// TwinCAT 3 PLC project PLC1
// ProgramVersion: 3.1.4026.24
// CompilerDefines: VISU_USEPROPERTYINFO
// libraries:
//   Tc2_Standard, * (Beckhoff Automation GmbH)
//   Tc2_System, * (Beckhoff Automation GmbH)
//   Tc2_TcpIp, * (Beckhoff Automation GmbH)
//   Tc2_Utilities, * (Beckhoff Automation GmbH)
//   VisuDialogs, * (System)
//   VisuSymbols,3.5.10.0,System
// project tree:
//   DUTs/ E_AutoStep.TcDUT (not stored), E_ControlMode.TcDUT, E_LogSev.TcDUT, E_MasterAutoStep.TcDUT, E_RobotConnState.TcDUT, ST_HmiMasterAuto.TcDUT, ST_HmiMasterAutoCfg.TcDUT, ST_HmiPiston.TcDUT (not stored), ST_HmiPistonAuto.TcDUT, ST_HmiPistonAutoCfg.TcDUT, ST_HmiRobot.TcDUT, ST_RobotParams.TcDUT, ST_LogEntry.TcDUT, E_LogFileState.TcDUT, ST_HmiLogFile.TcDUT, ST_HmiLogFileCfg.TcDUT
//   / GlobalTextList.TcGTLO, IOmapTask.TcTTO, PlcTask.TcTTO (not stored), VISU_TASK.TcTTO
//   GVLs/ GVL_App.TcGVL, GVL_HMI.TcGVL, GVL_HmiPersistent.TcGVL, GVL_IO.TcGVL (not stored), GVL_Log.TcGVL, GVL_Robot.TcGVL
//   POUs/ F_LogEvent.TcPOU, FB_PersistentAutoSave.TcPOU, FB_LogCsvWriter.TcPOU, FB_MasterAutoCycle.TcPOU, FB_PistonAutoCycle.TcPOU (not stored), FB_RobotTcpClient.TcPOU, FB_SolSolPiston_2Pos.TcPOU, FB_SolSpringPiston_2Pos.TcPOU, MAIN.TcPOU, PRG_IoMap.TcPOU
//   VISU/ Main.TcVIS, PistonsManual.TcVIS, Logs.TcVIS, Robot.TcVIS, GripperManual.TcVIS, Piston.TcVIS, AutoMain.TcVIS, AutoConfig.TcVIS, VisualizationManager.TcVMO (not stored)
// real-time tasks:
//   TASK IOmapTask: cycle T#5ms, priority 15, ADS port 350
//   TASK PlcTask: cycle T#10ms, priority 20, ADS port 351
//   TASK VISU_TASK: cycle T#200000us, priority 30, ADS port 352
// I/O:
//   DEVICE Device 1 (EtherCAT), AmsNetId 5.79.93.36.2.1
//     Term 1 (EK1100) [EK1100 EtherCAT Coupler (2A E-Bus)]
//       Term 2 (EL1809) [EL1809 16Ch. Dig. Input 24V, 3ms]
//       Term 3 (EL1008) [EL1008 8Ch. Dig. Input 24V, 3ms]
//       Term 4 (EL2809) [EL2809 16Ch. Dig. Output 24V, 0.5A]
//       Term 5 (EL9011) [EL9011 End Terminal]
// variable links:
//   PLC1/PLC1 Instance <-> Device 1 (EtherCAT)/Term 1 (EK1100)/Term 2 (EL1809)
//     IOmapTask Inputs/GVL_IO.dIn[{1..16}] <-> Channel {1..16}/Input  (16 links)
//   PLC1/PLC1 Instance <-> Device 1 (EtherCAT)/Term 1 (EK1100)/Term 3 (EL1008)
//     IOmapTask Inputs/GVL_IO.dIn[{17..24}] <-> Channel {1..8}/Input  (8 links)
//   PLC1/PLC1 Instance <-> Device 1 (EtherCAT)/Term 1 (EK1100)/Term 4 (EL2809)
//     IOmapTask Outputs/GVL_IO.dOut[{1..16}] <-> Channel {1..16}/Output  (16 links)

CONFIGURATION PLC1
    RESOURCE PLC ON TwinCAT3
        TASK IOmapTask(INTERVAL := T#5ms, PRIORITY := 15);
        TASK VISU_TASK(INTERVAL := T#200000us, PRIORITY := 30);
        PROGRAM PRG_IoMap WITH IOmapTask : PRG_IoMap;
        PROGRAM VisuElems_Visu_Prg WITH VISU_TASK : VisuElems.Visu_Prg;
    END_RESOURCE
END_CONFIGURATION

// ---- DUTs/E_ControlMode.TcDUT
{attribute 'qualified_only'}
{attribute 'strict'}
{attribute 'to_string'}
TYPE E_ControlMode :
(
    Manual    := 0,
    Automatic := 1
) ;
END_TYPE

// ---- DUTs/E_LogSev.TcDUT
{attribute 'qualified_only'}
{attribute 'strict'}
{attribute 'to_string'}
TYPE E_LogSev :
(
    DBG   := 0,   // dropped by F_LogEvent when GVL_Log.bDebugMode = FALSE
    INFO  := 1,
    WARN  := 2,
    ERR   := 3
) ;
END_TYPE

// ---- DUTs/E_MasterAutoStep.TcDUT
{attribute 'qualified_only'}
{attribute 'strict'}
{attribute 'to_string'}
TYPE E_MasterAutoStep :
(
    IDLE                 := 0,
    SEP_EXTENDING        := 1,
    WAIT_POS2            := 2,
    PUSH_EXTENDING       := 3,
    DWELL_PUSH           := 4,
    PUSH_RETRACTING      := 5,
    PUSH_RETRACTED_DWELL := 6,
    SEP_RETRACTING       := 7,
    SEP_RETRACTED_DWELL  := 8,
    INIT_PUSH_RETRACTING := 10,
    INIT_SEP_RETRACTING  := 11,
    INIT_GRIP_RETRACTING := 12,
    // Renamed from WAIT_PLATE 2026-08-05. Wire value 20 is UNCHANGED, so the
    // robot cannot tell the difference; only the panel text and the source read
    // differently. It does more than wait -- it is the plate-presence gate.
    CHECK_PLATE          := 20,
    GRIP_EXTENDING       := 21,
    GRIP_RETRACTING      := 22,
    MANUAL               := 30,
    // In Automatic but NOT armed: the pistons have not been homed under
    // operator control since power-up / Manual / a STOP, so the robot must not
    // command a cycle. Exited only by an operator START (HMI button or PB3),
    // which runs the INIT retract chain and lands in IDLE.
    //
    // 40 sits in the same "not a sequence step" class as MANUAL(30) and
    // ERR(99). Values are WIRE values -- nStateOut is read by the robot -- so
    // nothing here may ever be renumbered.
    //
    // Keep the name short: sStepText is STRING(20) and INIT_PUSH_RETRACTING
    // already fills it exactly, so a longer enumerator would truncate.
    NOT_HOMED            := 40,

    // Fault-recovery retract chain, added 2026-08-05. Same MOTION as the
    // RETRACT/INIT chain (push, then sep, then grip -- the collision ordering)
    // but its own identity, so a failed recovery is distinguishable from a
    // failed arming: distinct sStepText, distinct error codes 12/13/14, and a
    // distinct value on the wire.
    //
    // Entered only from ERR on RESET; exits to IDLE (armed). 50/51/52 rather
    // than 13/14/15 because a fresh decade matches the convention that
    // non-bulb-cycle states own decades (30 Manual, 40 Not-homed, 99 Err), and
    // STATE:5x is instantly greppable in a robot log. Adjacency to 10/11/12
    // would invite exactly the confusion these states exist to remove.
    //
    // The robot needs NO new branch: it acts on 0 (armed), 99 (faulted) and
    // treats everything else as "wait", which is correct for all three.
    //
    // Names are <= 20 chars because sStepText is STRING(20).
    RECOVER_PUSH_RETR    := 50,
    RECOVER_SEP_RETR     := 51,
    RECOVER_GRIP_RETR    := 52,

    ERR                  := 99
) ;
END_TYPE

// ---- DUTs/E_RobotConnState.TcDUT
{attribute 'qualified_only'}
{attribute 'strict'}
{attribute 'to_string'}
TYPE E_RobotConnState :
(
    Disconnected := 0,
    Connecting   := 1,
    Connected    := 2,
    Error        := 3
) ;
END_TYPE

// ---- DUTs/ST_HmiMasterAuto.TcDUT
TYPE ST_HmiMasterAuto :
STRUCT
    // Display label ('MasterAuto'). Set from GVL_HMI init, never written by FB.
    Name             : STRING(30);

    // HMI writes -- momentary command buttons (R_TRIG inside FB latches the
    // rising edge). NOTE bStart means "home the pistons and arm", NOT "run a
    // bulb cycle" -- only the robot's CMD:1 starts a cycle. Also driven by the
    // green PB3 in Automatic (see MAIN).
    bStart           : BOOL;
    (* Operator "run ONE bulb from IDLE" -- the HMI parallel to holding the
       orange PB2 + green PB3 combo, and to the robot's CMD:1. Momentary:
       FB_MasterAutoCycle detects the rising edge and clears it.

       Deliberately a SEPARATE field from bStart. bStart means "home and
       arm" and is accepted in NOT_HOMED only; making it also mean "run a
       bulb" in IDLE would give one symbol two meanings that differ by
       state, which is exactly the shape that let a green-before-orange
       combo press silently lose its bulb request (fixed 2026-08-05 by
       removing START from IDLE -- do not put it back).

       Also separate from bSimStartAssembly, which is the documented BENCH
       stand-in for the robot. Two fields keep "an operator started a bulb"
       and "someone simulated the robot" distinguishable in the log ring. *)
    bStartCycle      : BOOL;
    bStop            : BOOL;
    bReset           : BOOL;

    // FB writes -- status.
    //
    // Defaults to NOT_HOMED, and that default is what keeps the machine still
    // after a power cycle: GVL_HMI is plain VAR_GLOBAL, so this initialiser is
    // re-applied on every cold boot and every download. bAutoMode persists, so
    // without it the panel would come back in Automatic reporting IDLE(0) and a
    // running robot could command a cycle with the pistons anywhere.
    eStep            : E_MasterAutoStep := E_MasterAutoStep.NOT_HOMED;
    sStepText        : STRING(20);   // human-readable mirror of eStep
    tElapsedS        : LREAL;        // seconds spent in the current step (0.0 on transition)
    iErrorCode       : INT;          // 0 = OK; see FB_MasterAutoCycle header for the code table
    sErrorText       : STRING(80);
    nCyclesCompleted : UDINT;        // incremented at end of GRIP_RETRACTING

    // HMI writes -- bench sim of the robot's start command. Rising edge inside
    // the FB behaves the same as an incoming CMD:1 pulse (see bExtStartPulse).
    // FB auto-clears this flag after the rising edge is consumed.
    bSimStartAssembly      : BOOL;

    // HMI writes -- per-step Simulate flags. Rising edge shortcuts the current
    // step's wait condition (FB clears the flag on consumption via R_TRIG.Q).
    bSimStep_Idle          : BOOL;
    bSimStep_InitPushRet   : BOOL;
    bSimStep_InitSepRet    : BOOL;
    bSimStep_InitGripRet   : BOOL;
    bSimStep_WaitPlate     : BOOL;
    bSimStep_GripExt       : BOOL;
    bSimStep_SepExt        : BOOL;
    bSimStep_WaitPos2      : BOOL;
    bSimStep_PushExt       : BOOL;
    bSimStep_DwellPush     : BOOL;
    bSimStep_PushRet       : BOOL;
    bSimStep_PushRetDwell  : BOOL;
    bSimStep_SepRet        : BOOL;
    bSimStep_SepRetDwell   : BOOL;
    bSimStep_GripRet       : BOOL;
    (* The RECOVER chain wants sim flags for the same reason the INIT chain
       has them: all three are sensor-waiting states, so without these a
       recovery cannot be stepped on a bench whose sensors are not wired.
       Added 2026-08-05; the RECOVER states themselves shipped without them. *)
    bSimStep_RecoverPushRet : BOOL;
    bSimStep_RecoverSepRet  : BOOL;
    bSimStep_RecoverGripRet : BOOL;
END_STRUCT
END_TYPE

// ---- DUTs/ST_HmiMasterAutoCfg.TcDUT
TYPE ST_HmiMasterAutoCfg :
STRUCT
    // Timers, milliseconds. UDINT so HMI NumericInput binds directly.
    tDwellPushMs            : UDINT := 2000;   // DWELL_PUSH -- hold at push-extended
    tPushRetractedDwellMs   : UDINT := 500;    // PUSH_RETRACTED_DWELL -- hold after push retract
    tSepRetractedDwellMs    : UDINT := 500;    // SEP_RETRACTED_DWELL -- hold after sep retract before IDLE

    // Timeout guards every non-DWELL waiting state. On expiry, iErrorCode is
    // set to the step's numeric code and the cycle enters ERR.
    tStepTimeoutMs          : UDINT := 10000;

    // Dedicated timeout for CHECK_PLATE (bounded by robot placement time, not
    // by a motion budget). On expiry, iErrorCode := 9 and the cycle enters ERR
    // — unless bBypassPlateSensors is set, see below.
    tPlateWaitTimeoutMs     : UDINT := 10000;

    // Panel push-button HOLD durations, milliseconds. Both are deliberate
    // two-hand / sustained gestures rather than edges, so a knock or a brushed
    // sleeve cannot trigger them.
    //
    // tPbStopHoldMs  — how long the RED PB1 must be held in Automatic to STOP
    //                  the machine (disarm to NOT_HOMED).
    // tPbStartHoldMs — how long the GREEN PB3 and ORANGE PB2 must be held
    //                  TOGETHER to start one bulb cycle from IDLE, which is the
    //                  operator's parallel to the robot's CMD:1.
    //
    // Editable on AutoMain so the duration can be tuned to the operators
    // without a rebuild.
    tPbStopHoldMs           : UDINT := 1000;
    tPbStartHoldMs          : UDINT := 1000;

    // If TRUE, the 4 movement states ignore sensor feedback and advance when
    // tStepTimeoutMs expires — the timeout doubles as the fixed step duration.
    // No timeout-error path while sensorless. Mirrors ST_HmiPistonAutoCfg.bNoSensors.
    // Deliberately does NOT cover WAIT_PLATE — use bBypassPlateSensors for that.
    bNoSensors              : BOOL  := FALSE;

    // Plate-sensor bypass. Removes only the WAIT_PLATE timeout ERROR, not the
    // wait itself: the bPlateSenL AND bPlateSenR fast-path still advances the
    // cycle as normal, so with healthy sensors nothing changes. With unwired
    // or faulty ones, tPlateWaitTimeoutMs degrades into a fixed placement
    // dwell and the cycle continues instead of raising error 9.
    // Separate from bNoSensors on purpose: skipping the plate gate is a
    // safety-relevant decision and should be made explicitly, not inherited
    // from a bench-testing flag.
    bBypassPlateSensors     : BOOL  := FALSE;

    // NOTE bAutoMode used to live here and does NOT any more (2026-08-06).
    // It moved to GVL_HMI.bAutoMode -- plain VAR_GLOBAL, initialised TRUE -- so
    // that every power-up comes back in Automatic instead of restoring whatever
    // mode the operator happened to leave selected. Persisting it was the older
    // decision (2026-07-27) and it had the property that a technician who
    // switched to Manual to jog a piston found the machine still in Manual after
    // a reboot; the machine's normal condition is Automatic, so that is now the
    // condition it boots into. It is safe because arming is separate: eStep still
    // defaults to NOT_HOMED, so nothing moves until someone presses ENABLE AUTO.
    //
    // This struct is now purely operator-tunable CONFIG -- timers and the two
    // bench flags -- which is also what makes it a coherent unit to put on its
    // own AutoConfig page.
END_STRUCT
END_TYPE

// ---- DUTs/ST_HmiPistonAuto.TcDUT
TYPE ST_HmiPistonAuto :
STRUCT
    // HMI writes — momentary commands (R_TRIG inside FB latches the rising edge)
    bStart : BOOL;
    bStop  : BOOL;
    bReset : BOOL;
    bAck   : BOOL;

    // FB writes — status (never touched by HMI)
    eStep            : E_AutoStep;
    sStepText        : STRING(20);   // human-readable mirror of eStep
    tElapsedS        : LREAL;        // seconds spent in the current step (0.0 on transition)
    bError           : BOOL;
    sErrorText       : STRING(80);
    nCyclesCompleted : UDINT;        // incremented at end of each DWELL_RET
END_STRUCT
END_TYPE

// ---- DUTs/ST_HmiPistonAutoCfg.TcDUT
TYPE ST_HmiPistonAutoCfg :
STRUCT
    // All times in milliseconds. UDINT so HMI NumericInput binds directly (no TIME<->UDINT juggling).

    // Dwell = how long to sit at the sensor before starting the reverse move.
    tDwellExtendedMs   : UDINT := 500;
    tDwellRetractedMs  : UDINT := 500;

    // Timeout = if we do not see the target sensor within this window, raise an error.
    tTimeoutExtendMs   : UDINT := 3000;
    tTimeoutRetractMs  : UDINT := 3000;

    // If TRUE, DWELL_RET loops back to EXTENDING instead of returning to IDLE.
    bContinuous        : BOOL  := FALSE;

    // If TRUE, the state machine ignores sensor feedback and advances on
    // timers alone: EXTENDING lasts tTimeoutExtendMs, RETRACTING lasts
    // tTimeoutRetractMs, then dwells run as usual. Use for bench cycling
    // when proximity switches aren't wired (SepSol2/3, PushSol2/3 today).
    // No feedback-mismatch check and no "sensor never arrived" error path.
    bNoSensors         : BOOL  := FALSE;
END_STRUCT
END_TYPE

// ---- DUTs/ST_HmiRobot.TcDUT
TYPE ST_HmiRobot :
STRUCT
    // Display label ('Robot'). Set from GVL_Robot, never written by bridge.
    Name           : STRING(30);

    // ------------------------------------------------------------------
    // Robot comms are now TCP-only. Start/reset commands come from the
    // robot as CMD:n replies (see ST_RobotParams.nRobotCmd); PLC state is
    // pushed to the robot as STATE:n (see ST_RobotParams.nStateOut). The
    // former discrete-I/O handshake (bStartAssembly/bAssemblyRunning wired
    // to STAND_SEQ_DO/STAND_SEQ_DI) is retired -- DI[13] and DO[7] are now
    // free channels.
    //
    // Fields below are the TCP status mirror written by FB_RobotTcpClient
    // and read by the HMI.
    // ------------------------------------------------------------------
    eConnState     : E_RobotConnState;
    sConnStateText : STRING(20);
    nPacketsRx     : UDINT;
    nPacketsTx     : UDINT;
    sLastMessage   : STRING(80);
    sLastTxMessage : STRING(80);

    // Consecutive failed connect attempts in the CURRENT outage; reset to 0 the
    // moment a connect succeeds. Added 2026-08-10 together with the edge guard on
    // the connect-failure log.
    //
    // THIS FIELD IS WHY THE SUPPRESSION IS SAFE. FB_RobotTcpClient re-dials every
    // ~3 s while bTcpEnable is TRUE, and it used to log an ERR every single time:
    // measured on the panel, all 20 slots of GVL_Log.aRecent were the same
    // 'Connect failed' line, and the Phase 2 CSV came out 95% that one message at
    // ~1.2 MB/day. Now only the first failure of an outage is logged (plus any
    // change of error NUMBER), so the information is not lost -- it moves here,
    // where the Robot page can show "312 failed attempts" in one field instead of
    // 312 log lines.
    nConnectFails  : UDINT;

    // The deprecated POS/AUTO_STARTED fields (bAtPos1/2/3, bTxAutoStarted,
    // bTxPushDone, bTxPistonsError, bRxResetError) were deleted 2026-07-26.
    // They existed only for legacy Flower_HMI page bindings on the retired
    // TCP POS protocol; that project is gone, no PLC code touched them, and
    // FlowerPyHmi does not poll them (scripts/check_pyhmi_contract.py).
END_STRUCT
END_TYPE

// ---- DUTs/ST_RobotParams.TcDUT
TYPE ST_RobotParams :
STRUCT
    // ------------------------------------------------------------------
    // Dobot tuning parameters exchanged over TCP:6001. TCP is now the ONLY
    // robot channel -- start/stop moved from discrete I/O to STATE:n / CMD:n
    // frames (see nStateOut / nRobotCmd below). Field names and order match
    // the robot's SYNC string (global.lua / dummy_server.py). Defaults
    // mirror the dummy server.
    //
    // UNITS AND RANGES. The four speeds are PERCENTAGES, not absolute
    // velocities: global.lua Init() passes J_SPEED / L_SPEED to VelJ() /
    // VelL(), and WAX_SPEED / WATER_SPEED feed the v= velocity-ratio option
    // of MovL. A global SpeedFactor(80) scales everything on top. The waits
    // are milliseconds. INT is an encoding detail, not a statement of range.
    //
    // Ranges below are the vendor's own -- the Dobot tuning GUI
    // (Robot\167-01-Saad\tcp client.py) clamps to them, and readme.txt
    // mirrors the table. The robot's Lua does NOT validate (src2.lua assigns
    // tonumber() straight through), so FB_RobotTcpClient.ClampParam enforces
    // them for every writer. The panel's NumericInputs also carry matching
    // InputBoxMin/Max, but per-control limits only bound their own control.
    // ------------------------------------------------------------------
    J_SPEED            : INT := 10;     //    1..100  %
    L_SPEED            : INT := 10;     //    1..100  %
    REPEATS            : INT := 2;      //    1..10
    START_WAIT         : INT := 500;    //   10..10000 ms
    WATER_WAIT         : INT := 500;    //   10..10000 ms
    STAND_WAIT         : INT := 2000;   //   10..10000 ms
    END_WAIT           : INT := 500;    //   10..10000 ms
    WATER_SPEED        : INT := 10;     //    0..100  %
    WAX_WAIT_TIME_IN   : INT := 500;    //    0..10000 ms
    WAX_WAIT_TIME_OUT  : INT := 500;    //   10..10000 ms
    WAX_SPEED          : INT := 10;     //    0..100  %

    // ------------------------------------------------------------------
    // Request flags -- FB_RobotTcpClient consumes each on the next idle
    // scan while Connected, sends the matching message, then auto-clears
    // the flag once the reply is received. Rising-level, not edge: setting
    // TRUE from the HMI is enough.
    // ------------------------------------------------------------------

    // Send GET_SYNC; the SYNC reply is parsed back into the 11 fields above.
    // The FB also raises this itself once, right after each (re)connect.
    bGetSync           : BOOL;

    // Raw escape hatch: send "sSetName:nSetVal" (e.g. "J_SPEED:15"); robot
    // replies "OK: SET NAME". NOT needed for the 11 params above -- writing
    // one of those fields directly (from the HMI or ST) is detected by
    // FB_RobotTcpClient's shadow-copy comparison and pushed automatically.
    // Use this only for names that are not fields of this struct.
    bSetParam          : BOOL;
    sSetName           : STRING(30);
    nSetVal            : INT;

    // Send "New_Bulb:1"; robot replies "OK: SET New_Bulb" and starts a fresh bulb.
    bTriggerNewBulb    : BOOL;

    // ------------------------------------------------------------------
    // State + command channel (replaces the retired discrete-I/O handshake).
    //
    // nStateOut : INT -- MAIN writes each scan. Value is TO_INT(eStep) in
    //   Automatic mode, or E_MasterAutoStep.MANUAL (30) when bAutoMode=FALSE.
    //   FB_RobotTcpClient sends "STATE:n" on change and every STATE_IDLE_MS
    //   as keep-alive.
    //
    // nRobotCmd : INT -- FB_RobotTcpClient writes each time a "CMD:n" reply
    //   carries a command. MAIN consumes it as a LEVEL (1 = start cycle,
    //   2 = reset error) and CLEARS it to 0 in the same scan; that clear is
    //   the PLC's acknowledgement, so the field normally reads 0 and a robot
    //   start is traced on the Logs page instead. The robot re-asserting the
    //   same value is therefore always honoured -- see the MAIN comment for
    //   the deadlock this replaced.
    // ------------------------------------------------------------------
    nStateOut          : INT;
    nRobotCmd          : INT;
END_STRUCT
END_TYPE

// ---- DUTs/ST_LogEntry.TcDUT
TYPE ST_LogEntry :
STRUCT
    // Wall-clock HH:MM:SS, stamped by F_LogEvent from GVL_Log.sNow (which
    // MAIN refreshes once a second from FB_LocalSystemTime). Added 2026-07-27
    // for the panel's Logs page, which has no drainer to stamp entries for it.
    //
    // This struct used to carry no timestamp on the reasoning that "Python
    // assigns wall-clock time when it drains the ring" — true, but that only
    // ever covered FlowerPyHmi. FlowerPyHmi still stamps its own arrival time
    // and ignores this field; the two do not have to agree, and sTime is the
    // more accurate of the two since it is taken at the moment of the event
    // rather than up to plc_ring_poll_ms later.
    //
    // Second resolution only. If sub-second ordering ever matters, add
    // nTick : UDINT rather than widening this string.
    sTime   : STRING(8);


    eSev    : E_LogSev;

    // Display mirror of eSev, set by F_LogEvent. Exists because the classic
    // VISU text output cannot resolve an enum to its enumerator name --
    // {attribute 'to_string'} only enables TO_STRING() in ST, it does not
    // teach the visualization anything. Same reason ST_HmiMasterAuto carries
    // sStepText next to eStep. FlowerPyHmi ignores this field; it renders
    // from eSev via its own SEV_NAMES map.
    // STRING(8), not STRING(4): the four current names top out at 4 chars,
    // but an exactly-sized string would silently truncate a longer one.
    sSevText : STRING(8);

    sSource : STRING(20);    // short instance name, e.g. 'SepSol1Auto'
    sMsg    : STRING(80);    // human-readable message
END_STRUCT
END_TYPE

// ---- DUTs/E_LogFileState.TcDUT
(*
   State of FB_LogCsvWriter (Phase 2 of docs/plans/log-csv-file.md).

   Declared in Phase 1, ahead of the FB that uses it, for the same reason the
   RECOVER_* wire values were reserved in one commit: the enum is the shared
   vocabulary between the PLC, the VISU page and FlowerPyHmi, so pinning the
   values once means the contract changes once.

   'to_string' is here for ST only. It does NOT make the classic VISU resolve an
   enumerator to its name -- that is settled in this project and is why
   ST_HmiLogFile carries an sStateText mirror. Binding eState to a VISU text
   output renders 0/1/2/3/4, which shipped wrong twice on the Logs page before
   being fixed on 2026-07-27.
*)
{attribute 'qualified_only'}
{attribute 'strict'}
{attribute 'to_string'}
TYPE E_LogFileState :
(
    // Logging disabled, or nothing pending. The resting state.
    OFF      := 0,

    // Entries buffered, waiting for the flush interval or a full buffer.
    BUFFER   := 10,

    // A flush is in flight. These three mirror the async chain rather than
    // being collapsed into one BUSY: if a write wedges, which of the three
    // it wedged in is the whole diagnostic, and there is no other way to see
    // it on a panel with no file viewer.
    OPENING  := 20,
    WRITING  := 21,
    CLOSING  := 22,

    // Rotation or retention work in progress (new day, size cap, or the
    // oldest-first delete sweep).
    ROTATING := 30,

    // A file operation failed. iErrorCode / sErrorText hold the detail and the
    // FB backs off on a timer rather than retrying every scan.
    FAILED   := 99
) ;
END_TYPE

// ---- DUTs/ST_HmiLogFile.TcDUT
(*
   Runtime status of the durable CSV log. Phase 1 of
   docs/plans/log-csv-file.md.

   Instanced as GVL_Log.stLogFile, i.e. VOLATILE -- GVL_Log is plain VAR_GLOBAL.
   That split is the point: the CONFIG persists (stLogFileCfg) and the STATUS
   does not. A persisted byte count or error text would be restored on the next
   boot describing a file the runtime has not opened, and a stale FAILED with a
   plausible error string is worse than no status at all.

   WHY THERE IS A STATUS STRUCT AT ALL. The CP6606 has no file viewer and no
   supported CPython, so nobody can look at the directory to see whether logging
   is working. Every question you would answer by looking at the filesystem has
   to be answerable from these fields instead: is it writing, to what, how big,
   how many files, has it lost anything, and if it stopped, why.
*)
TYPE ST_HmiLogFile :
STRUCT
    // Filename only, no directory -- sDir is already visible in the config and
    // repeating it here would just risk the two disagreeing.
    sCurrentFile      : STRING(40);

    // Bytes written to the current file. Compared against
    // uiMaxFileKB * 1024 to decide an in-day roll.
    uiBytesInFile     : UDINT;

    // CSV files currently in sDir, refreshed by the retention sweep.
    uiFilesOnDisk     : UDINT;

    // Entries the writer never got to see, because nWriteIdx advanced more than
    // the 256-slot ring holds while a flush was stalled.
    //
    // THIS FIELD IS THE WHOLE REASON THE DRAIN LOGIC IS ALLOWED TO SKIP. Losing
    // entries under a stall is unavoidable -- the ring is finite. Losing them
    // SILENTLY is not acceptable, so the count is published here and Phase 2
    // also emits one synthetic CSV row recording the gap, so the loss is visible
    // in the file itself and not only in a symbol nobody thought to read.
    udiEntriesDropped : UDINT;

    // Last file error. 0 = none. Latched until the next successful flush, so a
    // failure that has since cleared is still visible afterwards.
    iErrorCode        : UDINT;
    sErrorText        : STRING(80);

    eState            : E_LogFileState;

    // STRING mirror of eState. Required, not convenience: the classic VISU
    // cannot stringify an enum, so a text output bound to eState renders the
    // raw number. Every enum in this project carries such a mirror for exactly
    // this reason -- sStepText, sErrorText, sConnStateText, sSevText.
    sStateText        : STRING(12);
END_STRUCT
END_TYPE

// ---- DUTs/ST_HmiLogFileCfg.TcDUT
(*
   Operator-tunable config for the durable CSV log. Phase 1 of
   docs/plans/log-csv-file.md.

   Instanced as GVL_HmiPersistent.stLogFileCfg, i.e. VAR_GLOBAL PERSISTENT.
   Read the PERSISTENT DATA section of CLAUDE.md before adding a field here:
   PERSISTENT declares a durable storage CLASS, not an automatic save, and it is
   FB_PersistentAutoSave that actually flushes it ~2 s after edits stop. A new
   field is invisible to that FB until it is added to the shadow compare.

   COLD-BOOT DECISION, which CLAUDE.md requires for every new persistent field:
   NOTHING HERE IS CLEARED in MAIN's cold-boot block. Every field is operator or
   commissioning config, so surviving a power cycle is the entire point. Contrast
   the machine-state fields, where a persisted value can move pistons on power-up
   and which is why that block exists at all. Nothing here can start a motion.

   PER-FIELD COMMENTS IN THIS STRUCT MUST STAY SHORT -- put the prose in
   docs/plans/log-csv-file.md instead. This block, being the TYPE's comment, is
   free; a MEMBER's comment is not. TwinCAT ships a symbol's declaration comment
   inside its ADS symbol-info reply, and pyads' receive buffer is 798 bytes.
   sDir's original ~2.8 kB comment produced a 2967-byte reply, which fails
   symbol-info resolution -- and because read_list_by_name resolves every name
   in a sum-up up front, that took the field out of FlowerPyHmi's batched poll
   and onto an individual round trip: +88 ms on a 100 ms cycle, /events 3.3 Hz
   -> 2.62 Hz, measured against this panel 2026-08-12. FlowerPyHmi caps how many
   such symbols it will carry (5), and three others in this project are already
   spending that budget: GVL_HMI.bAutoMode (1400 B),
   GVL_Robot.stParams.nStateOut (991 B) and GVL_Robot.stRobot.nConnectFails
   (817 B).

   So the rule is not "write less"; it is "write it where an ADS client will not
   have to download it 10 times a second."
*)
TYPE ST_HmiLogFileCfg :
STRUCT
    // DEFAULT OFF, deliberately. The panel boots from Compact Flash and CF has
    // a finite erase budget -- the reason FB_PersistentAutoSave debounces its
    // own writes rather than saving on every keystroke. A machine that never
    // needs the file log should never spend flash on it, so writing to the card
    // is an explicit opt-in rather than something inherited from a download.
    bEnabled      : BOOL := FALSE;

    // Directory, WITH a trailing backslash; the writer appends the filename.
    // MUST stay under '\Hard Disk\': '\Temp\' and the device root are the WinCE
    // RAM object store and do not survive a restart. Never fall back to them.
    // Reasoning, measurements and the two rules: docs/plans/log-csv-file.md.
    // KEEP SHORT -- this comment ships in the ADS symbol-info reply (798 B cap);
    // oversized, it drops sDir out of FlowerPyHmi's batched poll. See below.
    sDir          : STRING(80) := '\Hard Disk\Logs\';

    // Roll to a new file part within the day if one file passes this. A guard
    // against a fault storm producing a single unwieldy file, not the primary
    // rotation trigger -- that is the date.
    uiMaxFileKB   : UDINT := 512;

    // Total ceiling for the directory. Phase 3 deletes oldest-first until the
    // sum is under this. 16 MB of INFO-level CSV is months of normal running.
    uiMaxTotalMB  : UDINT := 16;

    // Buffer flush interval. THE FLASH-WEAR CONTROL: entries accumulate in RAM
    // and reach the card once per interval, so a busy second costs one write
    // rather than dozens. Do not "improve" this into a write-per-entry -- that
    // is the change this comment exists to prevent.
    uiFlushSec    : UDINT := 10;
END_STRUCT
END_TYPE

// ---- GVLs/GVL_App.TcGVL
{attribute 'qualified_only'}
// Cooked IO aliases. Bound to the raw GVL_IO.dIn[i]/dOut[i] hardware arrays
// in MAIN's read-inputs / write-outputs bookends. No AT %*: these are plain
// BOOLs the FBs consume — the actual hardware wiring lives in GVL_IO.
//
// Tag convention: <Device>Sol<N>  = single EXTEND coil (SOL-Spring).
// The mechanical spring returns the actuator when the coil is de-energised,
// so no per-actuator Retract alias exists. DI still has a Retracted sensor.
//
//   SepSolN : Pin separator N   (DI 1..6, DO 1..3)
//   PushSolN: Pin push N        (DI 7..12, DO 4..6)
//   PbN / LedPbN: panel push buttons + status LEDs (DI 13..15, DO 7..9).
//                Behavior mode-gated -- see field comments below.
//   GripSolL / GripSolR: side grip pistons that clamp the robot-placed plate
//                       (DI 17..20, DO 10..11)
//   PlateSenL / PlateSenR: plate-presence sensors gating cycle start
//                         (DI 21..22)
//
// DI layout (rewired 2026-07-27 to match the physical terminals):
//   dIn[1..6]   = SepSol1..3 (Retract, Extend)
//   dIn[7..12]  = PushSol1..3 (Retract, Extend)
//   dIn[13..15] = PB1/2/3
//   dIn[16]     = free -- spare channel closing out the second 8-ch terminal,
//                 so the grip sensors start on a terminal boundary
//   dIn[17..18] = GripSolL (Retract, Extend)
//   dIn[19..20] = GripSolR (Retract, Extend)
//   dIn[21..22] = PlateSenL / PlateSenR
//   dIn[23..24] = free
//
// DO layout:
//   dOut[1..3]   = SepSolN Extend
//   dOut[4..6]   = PushSolN Extend
//   dOut[7..9]   = PB1/2/3 LEDs
//   dOut[10..11] = GripSolL/R Extend
//   dOut[12]     = LED_GREEN (machine status)
//   dOut[13]     = LED_RED (machine status)
//   dOut[14..16] = free
VAR_GLOBAL
    // SepSol1 (Pin separator 1) — DI 1..2, DO 1
    bSensorSepRetracted1  : BOOL;
    bSensorSepExtended1   : BOOL;
    bValveSepExtend1      : BOOL;

    // SepSol2 (Pin separator 2) — DI 3..4, DO 2
    bSensorSepRetracted2  : BOOL;
    bSensorSepExtended2   : BOOL;
    bValveSepExtend2      : BOOL;

    // SepSol3 (Pin separator 3) — DI 5..6, DO 3
    bSensorSepRetracted3  : BOOL;
    bSensorSepExtended3   : BOOL;
    bValveSepExtend3      : BOOL;

    // PushSol1 (Pin push 1) — DI 7..8, DO 4
    bSensorPushRetracted1 : BOOL;
    bSensorPushExtended1  : BOOL;
    bValvePushExtend1     : BOOL;

    // PushSol2 (Pin push 2) — DI 9..10, DO 5
    bSensorPushRetracted2 : BOOL;
    bSensorPushExtended2  : BOOL;
    bValvePushExtend2     : BOOL;

    // PushSol3 (Pin push 3) — DI 11..12, DO 6
    bSensorPushRetracted3 : BOOL;
    bSensorPushExtended3  : BOOL;
    bValvePushExtend3     : BOOL;

    // GripSolL (side grip, left) — DI 17..18, DO 10
    bSensorGripRetractedL : BOOL;
    bSensorGripExtendedL  : BOOL;
    bValveGripExtendL     : BOOL;

    // GripSolR (side grip, right) — DI 19..20, DO 11
    bSensorGripRetractedR : BOOL;
    bSensorGripExtendedR  : BOOL;
    bValveGripExtendR     : BOOL;

    // Plate-presence sensors — DI 21..22 (input only; no coil)
    bPlateSenL : BOOL;
    bPlateSenR : BOOL;

    // Panel push buttons + status LEDs — DI 13..15 / DO 7..9.
    // PB1 in Auto  = cycle-start bypass (bypass of robot's CMD:1).
    // PB1 in Manual = hold to extend both grip pistons.
    // PB2 in Manual = hold to extend all 3 SepSol pistons.
    // PB3 in Manual = hold to extend all 3 PushSol pistons.
    // LEDs mirror the corresponding PB press state (wiring diagnostic).
    bPb1     : BOOL;
    bPb2     : BOOL;
    bPb3     : BOOL;

    // Machine status lamps -- DO 12 / DO 13. Driven by MAIN from the master
    // cycle's state, NOT press mirrors like the PB LEDs above.
    //   bLedRed   = master cycle latched in ERR.
    //   bLedGreen = Auto+IDLE steady, Auto+cycling blink, otherwise off.
    bLedGreen : BOOL;
    bLedRed   : BOOL;
    bLedPb1  : BOOL;
    bLedPb2  : BOOL;
    bLedPb3  : BOOL;
END_VAR

// ---- GVLs/GVL_HMI.TcGVL
{attribute 'qualified_only'}
{attribute 'TcHmiSymbol.AddSymbol'}
VAR_GLOBAL
    stSepSol1  : ST_HmiPiston := (Name := 'SepSol1');
    stSepSol2  : ST_HmiPiston := (Name := 'SepSol2');
    stSepSol3  : ST_HmiPiston := (Name := 'SepSol3');
    stPushSol1 : ST_HmiPiston := (Name := 'PushSol1');
    stPushSol2 : ST_HmiPiston := (Name := 'PushSol2');
    stPushSol3 : ST_HmiPiston := (Name := 'PushSol3');
    stGripSolL : ST_HmiPiston := (Name := 'GripSolL');
    stGripSolR : ST_HmiPiston := (Name := 'GripSolR');

    // Runtime state for the per-piston auto sequencers. Config for each
    // lives in the matching stXxxAutoCfg in GVL_HmiPersistent (PERSISTENT).
    // In this panel solution the master cycle is the sole auto driver;
    // these per-piston Auto structs exist so the HMI's UC_PistonAuto tiles
    // have something to bind to. Their bStart/bStop/bReset are effectively
    // no-ops in the 167_01 solution.
    stSepSol1Auto  : ST_HmiPistonAuto;
    stSepSol2Auto  : ST_HmiPistonAuto;
    stSepSol3Auto  : ST_HmiPistonAuto;
    stPushSol1Auto : ST_HmiPistonAuto;
    stPushSol2Auto : ST_HmiPistonAuto;
    stPushSol3Auto : ST_HmiPistonAuto;
    stGripSolLAuto : ST_HmiPistonAuto;
    stGripSolRAuto : ST_HmiPistonAuto;

    // Plate-presence sensors exposed to the HMI (indicator lamps on the
    // AutoCycle page). Mirror of GVL_App.bPlateSen* driven in MAIN.
    bPlateSenL : BOOL;
    bPlateSenR : BOOL;

    // Runtime state for the master (multi-piston + robot-coordinated) auto
    // sequence. Config for it lives in GVL_HmiPersistent.stMasterAutoCfg.
    stMasterAuto   : ST_HmiMasterAuto := (Name := 'MasterAuto');

    // Global machine mode — the single source of truth for every piston's mode.
    // FALSE = Manual (operator jogs each piston; the master cycle is held in
    // NOT_HOMED). TRUE = Automatic (FB_MasterAutoCycle owns all eight pistons).
    // MAIN enforces it every scan onto each piston's eMode AND bMode, so there
    // is no per-piston double-control -- "no option to double control".
    //
    // DELIBERATELY NOT PERSISTENT, and deliberately not in stMasterAutoCfg
    // (moved out of it 2026-08-06). This GVL is plain VAR_GLOBAL, so the
    // initialiser below is re-applied on every cold boot and every download:
    // the machine always comes up in Automatic, which is its normal condition,
    // rather than restoring whatever mode was last selected.
    //
    // Safe because arming is a separate axis: stMasterAuto.eStep defaults to
    // NOT_HOMED, which reports STATE:40 -- the robot reads that as "wait" -- so
    // nothing can move until an operator presses ENABLE AUTO. Booting Automatic
    // decides WHO may drive the pistons, not WHETHER they may move.
    //
    // Consequence worth knowing: a technician who selects Manual to jog a piston
    // and then power-cycles comes back in Automatic, where the PB jogs are off by
    // design. Re-select Manual after a reboot.
    // BOOL rather than E_ControlMode so the classic VISU binds a checkbox
    // directly, matching the per-piston bMode convention.
    bAutoMode      : BOOL := TRUE;
	// Bench soak (log-file testing): self-arm and restart a bulb on every IDLE.
	// Inert unless FB_MasterAutoCycle.bBenchBuild is TRUE -- a rebuild, not a
	// runtime switch. Reasoning is on that constant, not here.
	bTempTestContinuesAutoRun : BOOL := FALSE;
END_VAR

// ---- GVLs/GVL_HmiPersistent.TcGVL
{attribute 'qualified_only'}
{attribute 'TcHmiSymbol.AddSymbol'}
VAR_GLOBAL PERSISTENT
    // Auto-cycle configuration. PERSISTENT so operator-tuned dwell / timeout
    // values survive an Activate Configuration + PLC restart. Values reset
    // to the struct defaults only on a full cold-boot reset.
    stSepSol1AutoCfg  : ST_HmiPistonAutoCfg;
    stSepSol2AutoCfg  : ST_HmiPistonAutoCfg;
    stSepSol3AutoCfg  : ST_HmiPistonAutoCfg;
    stPushSol1AutoCfg : ST_HmiPistonAutoCfg;
    stPushSol2AutoCfg : ST_HmiPistonAutoCfg;
    stPushSol3AutoCfg : ST_HmiPistonAutoCfg;
    stGripSolLAutoCfg : ST_HmiPistonAutoCfg;
    stGripSolRAutoCfg : ST_HmiPistonAutoCfg;

    // Config for the master (multi-piston + robot-coordinated) auto sequence.
    // See ST_HmiMasterAutoCfg for the tunable list; defaults land on cold-boot.
    stMasterAutoCfg   : ST_HmiMasterAutoCfg;

    // Durable CSV log config -- Phase 1 of docs/plans/log-csv-file.md.
    // Default bEnabled = FALSE, so adding this changes no behaviour until an
    // operator turns it on. FB_PersistentAutoSave watches it explicitly; a
    // field added here is NOT flushed until it is in that FB's shadow compare.
    //
    // ADDING A FIELD TO THIS GVL CHANGES THE PERSISTENT LAYOUT, which can
    // invalidate the existing Port_851.bootdata. After the first download,
    // check that the operator's timers still hold their values -- if they have
    // fallen back to declared defaults, re-enter them once. Verified before this
    // change that the values WERE surviving (tStepTimeoutMs read 1000, not its
    // declared 10000), so a reset afterwards is attributable to this edit.
    stLogFileCfg      : ST_HmiLogFileCfg;
END_VAR

// ---- GVLs/GVL_Log.TcGVL
{attribute 'qualified_only'}
{attribute 'TcHmiSymbol.AddSymbol'}
VAR_GLOBAL
    // Ring buffer of the most recent log entries the PLC has produced.
    // The Python bridge polls nWriteIdx via ADS and drains new slots.
    //   write slot at any moment = (nWriteIdx MOD 256)
    //   overflow detected when (nWriteIdx - lastReadIdx) > 256
    aLog        : ARRAY[0..255] OF ST_LogEntry;

    // Monotonic write counter (never wraps in practice — UDINT overflows
    // after 2^32 writes ≈ 4.3 billion, decades even at 1 kHz logging).
    nWriteIdx   : UDINT;

    // Global mute for PLC-side logging. When FALSE, F_LogEvent early-returns
    // without writing to aLog or aRecent. HMI Logs page binds this.
    bLogEnabled : BOOL := TRUE;

    // Runtime toggle for DEBUG severity. F_LogEvent drops DBG entries
    // when this is FALSE. Operator can flip it from the HMI without a
    // rebuild. HMI ToggleSwitch on the Robot page binds here.
    bDebugMode  : BOOL := FALSE;

    // Newest-first mirror of the last 20 entries. F_LogEvent shifts the
    // slots down and writes aRecent[0] on every accepted call, so the HMI
    // Logs page can bind aRecent[0..19] directly in display order.
    // aRecent[0] is the newest entry.
    aRecent     : ARRAY[0..19] OF ST_LogEntry;

    // Wall-clock HH:MM:SS, refreshed once a second by MAIN from
    // FB_LocalSystemTime, and copied into every entry by F_LogEvent.
    // It lives here rather than inside F_LogEvent because a FUNCTION cannot
    // own the FB instance FB_LocalSystemTime needs — functions are stateless,
    // so the cyclic tick has to happen in a POU that has one.
    // Reads '--:--:--' until the time source reports valid, so a panel with
    // an unset RTC shows that plainly instead of a plausible wrong time.
    sNow        : STRING(8) := '--:--:--';

    // Wall-clock date YYYY-MM-DD, refreshed by MAIN section 0a alongside sNow
    // but only when the DAY rolls over. Exists because filenames need a date
    // and sNow is HH:MM:SS only.
    //
    // Reads '0000-00-00' until the time source reports valid, and the writer
    // treats that as "no date" and falls back to flower-nodate.csv rather
    // than building a filename out of it. An unset panel RTC is a real
    // condition here, not a hypothetical -- sNow already has the same guard.
    // The sortable YYYY-MM-DD order is load-bearing for Phase 3: retention
    // deletes oldest-by-NAME, which is only correct because these sort
    // chronologically.
    sToday      : STRING(10) := '0000-00-00';

    // Durable CSV log status -- Phase 1 of docs/plans/log-csv-file.md.
    // VOLATILE on purpose (GVL_Log is plain VAR_GLOBAL): the config persists,
    // the status must not. A restored byte count or a stale FAILED with a
    // plausible error string would describe a file this runtime never opened.
    stLogFile   : ST_HmiLogFile;

    // NOTE stBridgeCfg / ST_LogBridgeCfg used to live here and are GONE
    // (2026-08-07). The field existed solely so the retired
    // RobotBridge/log_pump.py could publish its own logger configuration for an
    // HMI to render. The bridge was retired 2026-07-26 and nothing wrote the
    // struct after that, so it read as empty strings and zeros and made a
    // shipped FlowerPyHmi page render a visibly blank block. Removed from
    // FlowerPyHmi first, then from here -- that order matters, because deleting
    // the symbol while the poller still asks for it makes read_many log
    // "dropping N unresolvable symbol(s)", which looks like a real fault.
END_VAR

// ---- GVLs/GVL_Robot.TcGVL
{attribute 'qualified_only'}
{attribute 'TcHmiSymbol.AddSymbol'}
VAR_GLOBAL
    stRobot : ST_HmiRobot := (Name := 'Robot');

    // Robot tuning parameters, request flags, and the STATE/CMD channel --
    // all exchanged over TCP:6001 by FB_RobotTcpClient, which is the SOLE
    // robot channel (the discrete-I/O handshake was retired 2026-07-26).
    // The 11 tuning params are read/write: editing one here is detected by
    // the FB's shadow-copy comparison and pushed to the robot.
    stParams : ST_RobotParams;

    // Master enable for the TCP client. FALSE holds it disconnected.
    // Deliberately NOT persistent: a link disabled for a bench session
    // should come back enabled after a power cycle rather than leaving the
    // robot silently unreachable with no obvious reason why.
    bTcpEnable : BOOL := TRUE;
END_VAR

VAR_GLOBAL PERSISTENT
    // TCP client target. PLC dials the robot's server. Host is set by the
    // commissioner (robot IP); port matches global.lua.
    //
    // PERSISTENT because the correct value DIFFERS BETWEEN INSTALLATIONS --
    // that, not "does it reset on boot", is the test for whether something
    // is configuration. As plain VAR_GLOBAL these were re-applied from the
    // literals below on every Activate Configuration, download and reset,
    // silently discarding whatever the commissioner had typed on the Robot
    // page. Nothing reported an error: the write succeeded, the field really
    // did change, and it really was reverted later.
    //
    // The declared values are the FACTORY DEFAULT, applied only on a
    // first-ever boot or Reset Origin. FB_PersistentAutoSave flushes edits
    // to disk ~2 s after the operator stops typing.
    //
    // *** CHANGING THE LITERAL BELOW DOES NOT CHANGE A COMMISSIONED PANEL. ***
    // That is the whole point of the PERSISTENT block above: any panel that has
    // already booted keeps its stored value, so a new default reaches only a
    // fresh install or a Reset Origin. To retarget a panel that is already
    // running, type the address on the Robot page (FB_RobotTcpClient tears the
    // live session down and re-dials) or do Reset Origin to fall back to this.
    //
    // Declared here rather than in GVL_HmiPersistent so the symbol paths
    // GVL_Robot.sRobotHost / .nRobotPort are unchanged -- a GVL may hold
    // both a volatile and a persistent block.
    sRobotHost : STRING := '192.168.1.11';   // was 192.168.201.1 until 2026-07-29
    nRobotPort : UINT := 6001;
END_VAR

// ---- POUs/PRG_IoMap.TcPOU
PROGRAM PRG_IoMap
VAR
END_VAR

ReadInputs();
WriteOutputs();

ACTION ReadInputs:
(* ==========================================
   READ INPUTS — copy raw GVL_IO.dIn[] channels into named GVL_App aliases.
   Each SOL-Spring actuator has both a Retracted and an Extended proximity
   switch (spring retracts, coil extends; both end positions get sensors).
   ========================================== *)
GVL_App.bSensorSepRetracted1  := GVL_IO.dIn[3];
GVL_App.bSensorSepExtended1   := GVL_IO.dIn[4];
GVL_App.bSensorSepRetracted2  := GVL_IO.dIn[7];
GVL_App.bSensorSepExtended2   := GVL_IO.dIn[8];
GVL_App.bSensorSepRetracted3  := GVL_IO.dIn[11];
GVL_App.bSensorSepExtended3   := GVL_IO.dIn[12];
GVL_App.bSensorPushRetracted1 := GVL_IO.dIn[1];
GVL_App.bSensorPushExtended1  := GVL_IO.dIn[2];
GVL_App.bSensorPushRetracted2 := GVL_IO.dIn[5];
GVL_App.bSensorPushExtended2  := GVL_IO.dIn[6];
GVL_App.bSensorPushRetracted3 := GVL_IO.dIn[9];
GVL_App.bSensorPushExtended3  := GVL_IO.dIn[10];

(* Panel push buttons. Consumer logic lives in MAIN and is mode-gated:
   PB3 in Auto is the operator START (home + arm); PB1/PB2/PB3 jog the
   grip / Sep / Push groups in Manual, and also while latched in ERR. *)
GVL_App.bPb1 := GVL_IO.dIn[13];
GVL_App.bPb2 := GVL_IO.dIn[14];
GVL_App.bPb3 := GVL_IO.dIn[15];

(* Grip pistons  *)
GVL_App.bSensorGripRetractedL := GVL_IO.dIn[17];
GVL_App.bSensorGripExtendedL  := GVL_IO.dIn[18];
GVL_App.bSensorGripRetractedR := GVL_IO.dIn[19];
GVL_App.bSensorGripExtendedR  := GVL_IO.dIn[20];

(* Plate-presence sensors. NOTE: only ONE need be TRUE for WAIT_PLATE to
   advance the cycle into GRIP_EXTENDING -- FB_MasterAutoCycle computes
   bPlateOk as an OR, a field deviation kept because only one plate sensor is
   confirmed wired. It is not the documented AND.

   NOTE ALSO: docs/167_01_SAAD_PinPush_IO_List.xlsx assigns dIn[21] to
   PlateSensR and dIn[22] to PlateSensL -- the OPPOSITE of the two lines
   below. Harmless for the cycle gate while bPlateOk is an OR, but it means
   the L / R lamps on Main.TcVIS are mislabelled. Settle which physical side
   is which before swapping either end. *)
GVL_App.bPlateSenL := GVL_IO.dIn[21];
GVL_App.bPlateSenR := GVL_IO.dIn[22];
END_ACTION

ACTION WriteOutputs:
(* ==========================================
   WRITE OUTPUTS — copy named GVL_App aliases into raw GVL_IO.dOut[] channels.
   Single Extend coil per actuator (SOL-Spring, spring retracts).
   ========================================== *)
GVL_IO.dOut[4] := GVL_App.bValveSepExtend1;
GVL_IO.dOut[5] := GVL_App.bValveSepExtend2;
GVL_IO.dOut[6] := GVL_App.bValveSepExtend3;
GVL_IO.dOut[1] := GVL_App.bValvePushExtend1;
GVL_IO.dOut[2] := GVL_App.bValvePushExtend2;
GVL_IO.dOut[3] := GVL_App.bValvePushExtend3;

(* Panel push-button status LEDs — mirror driven by MAIN. *)
GVL_IO.dOut[7] := GVL_App.bLedPb1;
GVL_IO.dOut[8] := GVL_App.bLedPb2;
GVL_IO.dOut[9] := GVL_App.bLedPb3;

(* Grip piston extend coils. *)
GVL_IO.dOut[10] := GVL_App.bValveGripExtendL;
GVL_IO.dOut[11] := GVL_App.bValveGripExtendR;

(* Machine status lamps. Green = Auto idle steady / cycling blink;
   red = master cycle in ERR. Both driven by MAIN. *)
GVL_IO.dOut[12] := GVL_App.bLedGreen;
GVL_IO.dOut[13] := GVL_App.bLedRed;
END_ACTION

END_PROGRAM

// ---- POUs/MAIN.TcPOU
PROGRAM MAIN
VAR
    fbSepSol1  : FB_SolSpringPiston_2Pos;
    fbSepSol2  : FB_SolSpringPiston_2Pos;
    fbSepSol3  : FB_SolSpringPiston_2Pos;
    fbPushSol1 : FB_SolSpringPiston_2Pos;
    fbPushSol2 : FB_SolSpringPiston_2Pos;
    fbPushSol3 : FB_SolSpringPiston_2Pos;
    fbGripSolL : FB_SolSpringPiston_2Pos;
    fbGripSolR : FB_SolSpringPiston_2Pos;

    // Full-machine sequencer coordinating the 3 pairs of (SepSolN,
    // PushSolN) + the 2 grip pistons. In this panel solution the master
    // cycle is the ONLY auto driver — the per-piston auto tiles
    // (bench-only feature) are removed, so no OR-merge at the call sites.
    fbMasterAutoCycle : FB_MasterAutoCycle;

    // Robot TCP/IP client — TCP-only protocol on :6001. Carries tuning
    // params + New_Bulb + STATE/CMD (state push out, command in). The
    // former discrete-I/O handshake (STAND_SEQ_DO/DI) is retired.
    fbRobotTcp : FB_RobotTcpClient;

    // Robot TCP command channel (nRobotCmd: 0=none, 1=start cycle,
    // 2=reset error). Consumed as a LEVEL and cleared on consumption --
    // see the body for why edge-detecting it deadlocked the machine.
    // bRobotStartPulse is the resulting one-scan pulse handed to
    // fbMasterAutoCycle's bExtStartPulse.
    bRobotStartPulse : BOOL;

    // PB3 rising edge in Auto is the operator START: "home the pistons and arm
    // the machine". Drives stMasterAuto.bStart, the same field as the HMI
    // button. PB3 because it is the GREEN button (PB1 red, PB2 orange) and this
    // is the go-ahead; it used to be PB1.
    //
    // Note it drives bStart, NOT bSimStartAssembly. Under the arming model
    // START no longer runs a bulb cycle, and bSimStartAssembly keeps its own
    // distinct job as the bench stand-in for the robot's CMD:1.
    fbTrigPb3 : R_TRIG;

    // PB2 rising edge in Auto -- RESET, but only while latched in ERR.
    fbTrigPb2 : R_TRIG;

    // The two Automatic HOLD gestures (2026-08-05). Each TON's IN is the
    // gesture itself, so releasing the button resets the elapsed time; .Q is a
    // level, so each is edge-detected to fire once per press.
    //
    //   PB1 held  -> STOP (disarm to NOT_HOMED)
    //   PB2 + PB3 -> run one bulb from IDLE, the operator's parallel to CMD:1
    //
    // Durations come from GVL_HmiPersistent.stMasterAutoCfg so they are tunable
    // on AutoMain without a rebuild.
    tonPb1Stop    : TON;
    fbTrigPb1Stop : R_TRIG;
    tonPbCombo    : TON;
    fbTrigPbCombo : R_TRIG;

    // One-scan pulse from the PB2+PB3 combo, OR-merged with the robot's start
    // pulse into fbMasterAutoCycle.bExtStartPulse -- both mean "run one bulb".
    bComboStartPulse : BOOL;

    // Scratch copies of the global machine mode, computed once per scan and
    // fanned out to all eight pistons (both eMode and bMode) just below.
    bMachineAuto : BOOL;
    bManualMode  : BOOL;   // = NOT bMachineAuto; gates PB jogs
    eMachineMode : E_ControlMode;

    // Flushes GVL_HmiPersistent to disk once the operator stops editing.
    // PERSISTENT alone never wrote anything on a power cut -- see the FB
    // header. Called last so it sees this scan's final config values.
    fbPersistentSave : FB_PersistentAutoSave;

    // Drains GVL_Log's ring to a CSV file on the panel's Compact Flash.
    // Phase 2 of docs/plans/log-csv-file.md. Idle until an operator sets
    // GVL_HmiPersistent.stLogFileCfg.bEnabled -- default FALSE.
    fbLogCsv : FB_LogCsvWriter;

    // Status-lamp blink source. A self-resetting TON toggling a BOOL gives a
    // 50% duty cycle; the TON on its own only produces a one-scan pulse,
    // which would make the lamp flicker rather than blink.
    tonBlink : TON;
    bBlink   : BOOL;

    // Wall clock for the log timestamps. Lives here because F_LogEvent is a
    // FUNCTION and cannot own an FB instance. dwCycle is in SECONDS.
    fbLocalTime : Tc2_Utilities.FB_LocalSystemTime;
    nLastSec    : WORD := 16#FFFF;   // impossible value, forces a first build
    sHH, sMM, sSS : STRING(2);

    // Date parts for GVL_Log.sToday, rebuilt only on a day rollover.
    // nLastDay starts at an impossible day so the first valid scan builds it.
    nLastDay      : WORD := 16#FFFF;
    sYYYY         : STRING(4);
    sMon, sDay    : STRING(2);
END_VAR

(* ==========================================
   0. CONTINUOUS IS DISABLED ON THE REAL MACHINE
   Forced FALSE every scan, not merely cleared at boot. The production
   machine never free-runs: every cycle is started by the operator or by the
   robot's CMD:1. The checkbox was removed from AutoMain, but a VISU page is
   only one of several writers — FlowerPyHmi has its own Continuous checkbox
   on two pages and reaches the field over ADS — so the field itself has to
   be the enforcement point. Any write is overwritten within one scan.

   It USED to be load-bearing: the IDLE branch tested it as a level, so a TRUE
   here re-armed a cycle with nothing external gating it. That is no longer the
   case -- the arming-model change of 2026-07-29 removed it from IDLE's exit
   condition, and the FB now writes bContinuous ten times and reads it ZERO
   times. This force-clear is belt-and-braces, not the interlock. What actually
   prevents power-up motion is eStep's NOT_HOMED default, below.

   bAutoMode is deliberately NOT touched (operator decision, 2026-07-27): the
   panel comes back in Automatic after a power cycle, still needing a real
   start trigger.

   This block used to add that it therefore came back in IDLE reporting
   nStateOut = 0, so "a robot already running may request a cycle straight
   after power-up -- that is the intended production behaviour". SUPERSEDED
   2026-07-29 and no longer true in either half. stHmi.eStep now DEFAULTS to
   NOT_HOMED (40), and GVL_HMI is plain VAR_GLOBAL so that initialiser is
   re-applied on every cold boot and download. A persisted bAutoMode = TRUE
   brings the panel back in Automatic but UN-ARMED, reporting 40, which the
   robot answers CMD:0 (wait). An operator START is required before anything
   can move. bAutoMode persists; the arming does not. See the ARMING MODEL
   section in CLAUDE.md.

   The timers, bNoSensors and bBypassPlateSensors are untouched too — they
   are operator config and persisting them is the point of the flush.
   ========================================== *)

(* ==========================================
   0a. LOG WALL CLOCK
   Refreshes GVL_Log.sNow, which F_LogEvent stamps into every entry so the
   Logs page can show a Time column. Rebuilt only when the second actually
   rolls over — the string work is trivial but there is no reason to redo it
   100 times a second.

   bValid gates it: an unset RTC shows '--:--:--' rather than a plausible
   wrong time, which is the difference between "the clock is not set" and
   "these events happened at 00:00:03".
   ========================================== *)
fbLocalTime(bEnable := TRUE, dwCycle := 1);

IF NOT fbLocalTime.bValid THEN
    GVL_Log.sNow   := '--:--:--';
    // Same discipline as sNow: an unset RTC must look unset. The CSV writer
    // reads this sentinel and falls back to flower-nodate.csv rather than
    // naming a file after garbage.
    GVL_Log.sToday := '0000-00-00';
ELSIF fbLocalTime.systemTime.wSecond <> nLastSec THEN
    nLastSec := fbLocalTime.systemTime.wSecond;
    // RIGHT(CONCAT('0', n), 2) is the zero-pad: '7' -> '07', '17' -> '17'.
    sHH := RIGHT(CONCAT('0', WORD_TO_STRING(fbLocalTime.systemTime.wHour)), 2);
    sMM := RIGHT(CONCAT('0', WORD_TO_STRING(fbLocalTime.systemTime.wMinute)), 2);
    sSS := RIGHT(CONCAT('0', WORD_TO_STRING(fbLocalTime.systemTime.wSecond)), 2);
    GVL_Log.sNow := CONCAT(CONCAT(CONCAT(CONCAT(sHH, ':'), sMM), ':'), sSS);

    // Date only on a DAY rollover, nested inside the second check so it costs
    // one WORD compare a second rather than string work. YYYY-MM-DD because
    // Phase 3 deletes oldest-by-name and that is only correct while the names
    // sort chronologically.
    IF fbLocalTime.systemTime.wDay <> nLastDay THEN
        nLastDay := fbLocalTime.systemTime.wDay;
        sYYYY := RIGHT(CONCAT('000', WORD_TO_STRING(fbLocalTime.systemTime.wYear)), 4);
        sMon  := RIGHT(CONCAT('0', WORD_TO_STRING(fbLocalTime.systemTime.wMonth)), 2);
        sDay  := RIGHT(CONCAT('0', WORD_TO_STRING(fbLocalTime.systemTime.wDay)), 2);
        GVL_Log.sToday := CONCAT(CONCAT(CONCAT(CONCAT(sYYYY, '-'), sMon), '-'), sDay);
    END_IF
END_IF

(* ==========================================
   Master auto-cycle — coordinates the 3 pairs of (Sep,Push) pistons
   with the robot handshake. Called BEFORE the per-piston
   auto FBs and BEFORE the piston FBs so its bSepCmd* / bPushCmd*
   outputs feed forward this scan.
   Master reads bIs* from the piston stHmi structs — those carry the
   previous scan's values (100 µs lag, negligible for a physical
   machine).
   ========================================== *)
fbMasterAutoCycle.bSepIsExtended[1]   := GVL_HMI.stSepSol1.bIsExtended;
fbMasterAutoCycle.bSepIsExtended[2]   := GVL_HMI.stSepSol2.bIsExtended;
fbMasterAutoCycle.bSepIsExtended[3]   := GVL_HMI.stSepSol3.bIsExtended;
fbMasterAutoCycle.bSepIsRetracted[1]  := GVL_HMI.stSepSol1.bIsRetracted;
fbMasterAutoCycle.bSepIsRetracted[2]  := GVL_HMI.stSepSol2.bIsRetracted;
fbMasterAutoCycle.bSepIsRetracted[3]  := GVL_HMI.stSepSol3.bIsRetracted;
fbMasterAutoCycle.bPushIsExtended[1]  := GVL_HMI.stPushSol1.bIsExtended;
fbMasterAutoCycle.bPushIsExtended[2]  := GVL_HMI.stPushSol2.bIsExtended;
fbMasterAutoCycle.bPushIsExtended[3]  := GVL_HMI.stPushSol3.bIsExtended;
fbMasterAutoCycle.bPushIsRetracted[1] := GVL_HMI.stPushSol1.bIsRetracted;
fbMasterAutoCycle.bPushIsRetracted[2] := GVL_HMI.stPushSol2.bIsRetracted;
fbMasterAutoCycle.bPushIsRetracted[3] := GVL_HMI.stPushSol3.bIsRetracted;

(* Grip pistons — L=[1], R=[2]. *)
fbMasterAutoCycle.bGripIsExtended[1]  := GVL_HMI.stGripSolL.bIsExtended;
fbMasterAutoCycle.bGripIsExtended[2]  := GVL_HMI.stGripSolR.bIsExtended;
fbMasterAutoCycle.bGripIsRetracted[1] := GVL_HMI.stGripSolL.bIsRetracted;
fbMasterAutoCycle.bGripIsRetracted[2] := GVL_HMI.stGripSolR.bIsRetracted;

(* Plate-presence sensors gate the cycle at WAIT_PLATE. Wire the raw
   GVL_App copies straight into the master cycle. Also mirror them onto
   GVL_HMI so the classic VISU / web HMI indicator lamps can bind. *)
fbMasterAutoCycle.bPlateSenL := GVL_App.bPlateSenL;
fbMasterAutoCycle.bPlateSenR := GVL_App.bPlateSenR;
GVL_HMI.bPlateSenL := GVL_App.bPlateSenL;
GVL_HMI.bPlateSenR := GVL_App.bPlateSenR;

(* ==========================================
   ROBOT COMMAND CONSUMPTION (nRobotCmd, written by fbRobotTcp on each
   CMD:<n> reply -- see the fbRobotTcp call further down).

   Consumed as a LEVEL and CLEARED here. The PLC clearing the field is the
   acknowledgement; the robot zeroing it after the next state push is now
   belt-and-braces rather than load-bearing.

   This used to be a pair of R_TRIGs on nRobotCmd = 1 / = 2, and nothing on
   the PLC side ever reset the field. That deadlocked the machine
   (2026-07-28, found on the real machine): a CMD:1 arriving while the panel
   was in Manual or latched in ERR fired the edge, the FB's IDLE branch
   correctly refused it, and nRobotCmd stayed at 1 forever. The robot
   re-asserts CMD:1 in every STATE reply until it sees the panel leave IDLE
   -- but re-sending a value that is already 1 produces no rising edge. So
   the robot waited for a state change while the PLC waited for an edge that
   could never come, and the Robot page showed CMD:1 arriving happily the
   whole time.

   Clearing makes it self-healing. A request that cannot be honoured this
   scan is dropped, and the robot's next keep-alive re-asserts it ~1 s
   later. Repeat pulses are harmless: only FB_MasterAutoCycle's IDLE branch
   consumes bExtStartPulse, and it is gated on bMachineAuto.

   Diagnostic note: nRobotCmd now reads 0 almost always, because it is
   consumed within a scan of arriving. The trace of a robot start is the
   'External start pulse' entry on the Logs page, and stRobot.sLastMessage
   still shows the raw CMD frame.

   RESET is fanned into the HMI bReset flag so operator- and robot-initiated
   resets share one consumption path inside the FB.
   ========================================== *)
bRobotStartPulse := FALSE;

IF GVL_Robot.stParams.nRobotCmd = 1 THEN
    bRobotStartPulse             := TRUE;
    GVL_Robot.stParams.nRobotCmd := 0;
ELSIF GVL_Robot.stParams.nRobotCmd = 2 THEN
    GVL_HMI.stMasterAuto.bReset  := TRUE;
    GVL_Robot.stParams.nRobotCmd := 0;
END_IF

fbMasterAutoCycle(
    bExtStartPulse := bRobotStartPulse OR bComboStartPulse,
    bMachineAuto   := GVL_HMI.bAutoMode,
    stHmi          := GVL_HMI.stMasterAuto,
    stCfg          := GVL_HmiPersistent.stMasterAutoCfg,
    stRobot        := GVL_Robot.stRobot
);

(* Global Auto/Manual hard interlock. The machine-wide bAutoMode is the single
   source of truth for every piston's mode — driven unconditionally each scan
   onto BOTH eMode and bMode so a per-piston toggle cannot create a second
   control path (no double-control). FB_SolSpringPiston_2Pos edge-syncs
   bMode<->eMode, so forcing only one would let a stray toggle propagate for a
   scan; forcing both closes that gap. In Automatic the master cycle owns all
   six pistons; in Manual the operator jogs them and the cycle is held in IDLE. *)
bMachineAuto := GVL_HMI.bAutoMode;
eMachineMode := SEL(bMachineAuto, E_ControlMode.Manual, E_ControlMode.Automatic);
GVL_HMI.stSepSol1.eMode  := eMachineMode;  GVL_HMI.stSepSol1.bMode  := bMachineAuto;
GVL_HMI.stPushSol1.eMode := eMachineMode;  GVL_HMI.stPushSol1.bMode := bMachineAuto;
GVL_HMI.stSepSol2.eMode  := eMachineMode;  GVL_HMI.stSepSol2.bMode  := bMachineAuto;
GVL_HMI.stPushSol2.eMode := eMachineMode;  GVL_HMI.stPushSol2.bMode := bMachineAuto;
GVL_HMI.stSepSol3.eMode  := eMachineMode;  GVL_HMI.stSepSol3.bMode  := bMachineAuto;
GVL_HMI.stPushSol3.eMode := eMachineMode;  GVL_HMI.stPushSol3.bMode := bMachineAuto;
GVL_HMI.stGripSolL.eMode := eMachineMode;  GVL_HMI.stGripSolL.bMode := bMachineAuto;
GVL_HMI.stGripSolR.eMode := eMachineMode;  GVL_HMI.stGripSolR.bMode := bMachineAuto;

(* ==========================================
   Panel push buttons. PB1 is RED, PB2 ORANGE, PB3 GREEN, and the colours
   drive the assignment.

   IN MANUAL — all three are momentary jogs. Hold to extend, release to
   retract: PB1 grip, PB2 Sep, PB3 Push. Unchanged.

   IN AUTOMATIC — three operator gestures, no jogs at all (operator decision
   2026-08-05: manual moves belong in Manual mode, not in any Auto state):

   * PB1 (red), HELD for tPbStopHoldMs   -> STOP. Disarms to NOT_HOMED.
   * PB3 (green), rising edge            -> START. "Home the pistons and arm."
                                            Drives stMasterAuto.bStart, the
                                            same field as the HMI button.
   * PB2 + PB3 together, HELD for
     tPbStartHoldMs, from IDLE           -> run ONE bulb cycle. The operator's
                                            parallel to the robot's CMD:1.
   * PB2 (orange), rising edge, in ERR   -> RESET.

   Why the two multi-second holds: both are consequential (one stops the
   machine, one starts a bulb), and a hold cannot be triggered by a knock or a
   brushed sleeve the way an edge can. Durations are operator-tunable on
   AutoMain rather than compiled in.

   PB3-vs-combo disambiguation: the standalone START edge is suppressed while
   PB2 is pressed, so the combo does not fire START on the way in. Press ORANGE
   first, then GREEN.

   Green-first is NOT harmless, and it was measured rather than assumed. It
   fires a plain START, so the machine re-homes. bComboStartPulse is one scan
   and bExtStartPulse is consumed ONLY by the IDLE branch, so:
     - homing done inside the hold  -> pointless re-home, then the cycle runs
     - still homing when it expires -> pulse DROPPED, no cycle, and the R_TRIG
                                       will not re-offer it while held
   On the machine, with real strokes, the second is the case to expect. See the
   TODO in CLAUDE.md about latching the request instead of pulsing it.

   * LED1 mirrors the press, and BLINKS while the STOP hold is counting.
   * LED2 mirrors the press.
   * LED3 is a state prompt in Auto -- assigned further down, after bBlink.
   ========================================== *)
GVL_App.bLedPb2 := GVL_App.bPb2;
(* PB3's LED is no longer a press mirror in Auto -- it is the "press me to arm"
   prompt. Assigned further down, after bBlink is refreshed, so the blink is
   this scan's value rather than last scan's. *)

(* ==========================================
   Machine status lamps (DO 12 green / DO 13 red).
   Unlike the PB LEDs above, which are dumb press mirrors, these report
   machine state:

     RED   = the master cycle is in its latched ERR state.
     GREEN = Auto and IDLE        -> steady  (armed, waiting for a start)
             Auto and cycling     -> blink   (running)
             Manual, or in ERR    -> off

   Green is off in ERR so the two lamps never contradict each other: red on
   with green also lit would read as "faulted but running". Green is off in
   Manual because it means "the automatic cycle is live", which is precisely
   what Manual is not.

   Blink source is a self-resetting TON toggling bBlink, giving 400 ms on /
   400 ms off. Using tonBlink.Q directly would light the lamp for a single
   scan per period -- invisible.
   ========================================== *)
tonBlink(IN := NOT tonBlink.Q, PT := T#400MS);
IF tonBlink.Q THEN
    bBlink := NOT bBlink;
END_IF

GVL_App.bLedRed := (GVL_HMI.stMasterAuto.eStep = E_MasterAutoStep.ERR);

IF NOT bMachineAuto
   OR GVL_HMI.stMasterAuto.eStep = E_MasterAutoStep.ERR
   OR GVL_HMI.stMasterAuto.eStep = E_MasterAutoStep.NOT_HOMED THEN
    (* Off in NOT_HOMED as well as Manual/ERR: green means "the automatic cycle
       is live and armed", and an un-homed machine is precisely not that. PB3's
       own green LED is the "press me" signal in that state, so the two are not
       competing for the operator's attention. *)
    GVL_App.bLedGreen := FALSE;
ELSIF GVL_HMI.stMasterAuto.eStep = E_MasterAutoStep.IDLE THEN
    GVL_App.bLedGreen := TRUE;
ELSE
    GVL_App.bLedGreen := bBlink;
END_IF

(* ==========================================
   PANEL GESTURES IN AUTOMATIC
   fbMasterAutoCycle already ran this scan, so eStep is current here.

   Both hold timers are driven with IN := <gesture held AND in Auto>, so
   releasing the button -- or leaving Auto -- resets the elapsed time and the
   operator has to start the hold again. .Q is a LEVEL, true for as long as the
   hold persists, so each one is edge-detected to fire exactly once per press.
   ========================================== *)

(* --- PB1 held -> STOP ------------------------------------------------------
   Writes stMasterAuto.bStop, the same field as the HMI STOP button, so the FB's
   existing Section 2 override handles it: disarm to NOT_HOMED, no error code. *)
tonPb1Stop(IN := bMachineAuto AND GVL_App.bPb1,
           PT := UDINT_TO_TIME(GVL_HmiPersistent.stMasterAutoCfg.tPbStopHoldMs));
fbTrigPb1Stop(CLK := tonPb1Stop.Q);
IF fbTrigPb1Stop.Q THEN
    GVL_HMI.stMasterAuto.bStop := TRUE;
END_IF;

(* --- PB2 + PB3 held -> run one bulb ----------------------------------------
   Fed into the SAME bExtStartPulse input the robot's CMD:1 uses, because it
   means exactly the same thing: "run one bulb". The FB's IDLE branch is the
   only consumer, and it is gated on bMachineAuto, so this cannot start a cycle
   from NOT_HOMED or from ERR -- the arming model is untouched. *)
tonPbCombo(IN := bMachineAuto AND GVL_App.bPb2 AND GVL_App.bPb3,
           PT := UDINT_TO_TIME(GVL_HmiPersistent.stMasterAutoCfg.tPbStartHoldMs));
fbTrigPbCombo(CLK := tonPbCombo.Q);
bComboStartPulse := fbTrigPbCombo.Q;
IF bComboStartPulse THEN
    F_LogEvent(eSev := E_LogSev.INFO, sSource := 'MAIN',
               sMsg := 'PB2+PB3 held: operator bulb start');
END_IF;

(* --- PB2 in ERR -> RESET ---------------------------------------------------
   An edge, not a hold: the machine is already stopped and latched, so there is
   nothing for a stray press to interrupt. Writes the same bReset field as the
   HMI button and the robot's CMD:2. *)
fbTrigPb2(CLK := GVL_App.bPb2);
IF bMachineAuto AND fbTrigPb2.Q
   AND GVL_HMI.stMasterAuto.eStep = E_MasterAutoStep.ERR THEN
    GVL_HMI.stMasterAuto.bReset := TRUE;
END_IF;

(* --- PB1 LED: press mirror, blinking while the STOP hold counts ------------
   A hold-to-act button with no feedback is guesswork; the blink tells the
   operator the hold is being counted. Assigned after bBlink is refreshed so it
   is this scan's value. *)
IF bMachineAuto AND GVL_App.bPb1 AND NOT tonPb1Stop.Q THEN
    GVL_App.bLedPb1 := bBlink;
ELSE
    GVL_App.bLedPb1 := GVL_App.bPb1;
END_IF

(* --- PB3 LED: "press me to arm" prompt ------------------------------------
   Blinks while in Auto and un-homed, off otherwise in Auto. Falls back to a raw
   press mirror in Manual, where PB3 is the Push jog and the LED keeps its
   original wiring-diagnostic role. *)
IF bMachineAuto THEN
    GVL_App.bLedPb3 := (GVL_HMI.stMasterAuto.eStep = E_MasterAutoStep.NOT_HOMED) AND bBlink;
ELSE
    GVL_App.bLedPb3 := GVL_App.bPb3;
END_IF

(* --- PB3 edge -> START ----------------------------------------------------
   Suppressed while PB2 is pressed so the PB2+PB3 combo does not fire a START on
   its way in. Press ORANGE first, then GREEN -- green-first can silently lose
   the cycle request, see the header. *)
fbTrigPb3(CLK := GVL_App.bPb3);
IF bMachineAuto AND NOT GVL_App.bPb2 AND fbTrigPb3.Q THEN
    GVL_HMI.stMasterAuto.bStart := TRUE;
END_IF;

bManualMode := NOT bMachineAuto;

(* ==========================================
   Pin separators (SOL-Spring, 2 limit switches, single Extend coil).
   The master cycle is the only auto driver; in Manual the piston FB
   ignores bAutoCmd* and follows the operator's jog buttons instead.
   ========================================== *)
fbSepSol1(
    bAutoCmdExtend   := fbMasterAutoCycle.bSepCmdExtend[1],
    bAutoCmdRetract  := fbMasterAutoCycle.bSepCmdRetract[1],
    bJogExtend       := bManualMode AND GVL_App.bPb2,
    bSwitchExtended  := GVL_App.bSensorSepExtended1,
    bSwitchRetracted := GVL_App.bSensorSepRetracted1,
    stHmi            := GVL_HMI.stSepSol1,
    bOutSolenoid     => GVL_App.bValveSepExtend1
);

fbSepSol2(
    bAutoCmdExtend   := fbMasterAutoCycle.bSepCmdExtend[2],
    bAutoCmdRetract  := fbMasterAutoCycle.bSepCmdRetract[2],
    bJogExtend       := bManualMode AND GVL_App.bPb2,
    bSwitchExtended  := GVL_App.bSensorSepExtended2,
    bSwitchRetracted := GVL_App.bSensorSepRetracted2,
    stHmi            := GVL_HMI.stSepSol2,
    bOutSolenoid     => GVL_App.bValveSepExtend2
);

fbSepSol3(
    bAutoCmdExtend   := fbMasterAutoCycle.bSepCmdExtend[3],
    bAutoCmdRetract  := fbMasterAutoCycle.bSepCmdRetract[3],
    bJogExtend       := bManualMode AND GVL_App.bPb2,
    bSwitchExtended  := GVL_App.bSensorSepExtended3,
    bSwitchRetracted := GVL_App.bSensorSepRetracted3,
    stHmi            := GVL_HMI.stSepSol3,
    bOutSolenoid     => GVL_App.bValveSepExtend3
);

(* ==========================================
   Pin pushers
   ========================================== *)
fbPushSol1(
    bAutoCmdExtend   := fbMasterAutoCycle.bPushCmdExtend[1],
    bAutoCmdRetract  := fbMasterAutoCycle.bPushCmdRetract[1],
    bJogExtend       := bManualMode AND GVL_App.bPb3,
    bSwitchExtended  := GVL_App.bSensorPushExtended1,
    bSwitchRetracted := GVL_App.bSensorPushRetracted1,
    stHmi            := GVL_HMI.stPushSol1,
    bOutSolenoid     => GVL_App.bValvePushExtend1
);

fbPushSol2(
    bAutoCmdExtend   := fbMasterAutoCycle.bPushCmdExtend[2],
    bAutoCmdRetract  := fbMasterAutoCycle.bPushCmdRetract[2],
    bJogExtend       := bManualMode AND GVL_App.bPb3,
    bSwitchExtended  := GVL_App.bSensorPushExtended2,
    bSwitchRetracted := GVL_App.bSensorPushRetracted2,
    stHmi            := GVL_HMI.stPushSol2,
    bOutSolenoid     => GVL_App.bValvePushExtend2
);

fbPushSol3(
    bAutoCmdExtend   := fbMasterAutoCycle.bPushCmdExtend[3],
    bAutoCmdRetract  := fbMasterAutoCycle.bPushCmdRetract[3],
    bJogExtend       := bManualMode AND GVL_App.bPb3,
    bSwitchExtended  := GVL_App.bSensorPushExtended3,
    bSwitchRetracted := GVL_App.bSensorPushRetracted3,
    stHmi            := GVL_HMI.stPushSol3,
    bOutSolenoid     => GVL_App.bValvePushExtend3
);

(* ==========================================
   Grip pistons — side clamps (L=[1], R=[2]) that hold the plate placed
   by the robot for the duration of the Sep/Push cycle.
   ========================================== *)
fbGripSolL(
    bAutoCmdExtend   := fbMasterAutoCycle.bGripCmdExtend[1],
    bAutoCmdRetract  := fbMasterAutoCycle.bGripCmdRetract[1],
    bJogExtend       := bManualMode AND GVL_App.bPb1,
    bSwitchExtended  := GVL_App.bSensorGripExtendedL,
    bSwitchRetracted := GVL_App.bSensorGripRetractedL,
    stHmi            := GVL_HMI.stGripSolL,
    bOutSolenoid     => GVL_App.bValveGripExtendL
);

fbGripSolR(
    bAutoCmdExtend   := fbMasterAutoCycle.bGripCmdExtend[2],
    bAutoCmdRetract  := fbMasterAutoCycle.bGripCmdRetract[2],
    bJogExtend       := bManualMode AND GVL_App.bPb1,
    bSwitchExtended  := GVL_App.bSensorGripExtendedR,
    bSwitchRetracted := GVL_App.bSensorGripRetractedR,
    stHmi            := GVL_HMI.stGripSolR,
    bOutSolenoid     => GVL_App.bValveGripExtendR
);

(* ==========================================
   Robot TCP/IP client (TCP-only protocol, port 6001). Runs every scan;
   its internal state machine dials the robot server and auto-reconnects
   on drop. The former discrete-I/O handshake is retired -- start/reset
   commands arrive via CMD:<n> replies, PLC state pushes via STATE:<n>.

   Compute nStateOut immediately after the master cycle so any transition
   this scan is visible to the robot on the next STATE push. MANUAL(30)
   sentinel while bAutoMode=FALSE so the robot knows the panel is out of
   auto and won't issue CMD:1.
   ========================================== *)
IF NOT GVL_HMI.bAutoMode THEN
    GVL_Robot.stParams.nStateOut := INT#30;   (* MANUAL *)
ELSE
    GVL_Robot.stParams.nStateOut := TO_INT(GVL_HMI.stMasterAuto.eStep);
END_IF

fbRobotTcp(
    bEnable     := GVL_Robot.bTcpEnable,
    sRemoteHost := GVL_Robot.sRobotHost,
    nRemotePort := GVL_Robot.nRobotPort,
    stRobot     := GVL_Robot.stRobot,
    stParams    := GVL_Robot.stParams
);

(* ==========================================
   Persistent config flush. Called LAST so it compares this scan's final
   values, and after section 0 so the cold-boot clears are part of its
   baseline rather than looking like an operator edit.
   Writes ~2 s after the operator stops editing; logs each flush to
   GVL_Log (visible on the Logs page) so a failing write is not silent.
   ========================================== *)
fbPersistentSave();

(* ==========================================
   Durable CSV log. Drains GVL_Log's 256-entry ring to a file on the Compact
   Flash. LAST in MAIN, after the persistent flush, so it sees every entry this
   scan produced -- including the flush's own log line.
   Does nothing until stLogFileCfg.bEnabled is set; default is FALSE, because
   the panel boots from CF and spending flash on logging is an explicit choice.
   ========================================== *)
fbLogCsv();

END_PROGRAM

// ---- POUs/FB_SolSpringPiston_2Pos.TcPOU
FUNCTION_BLOCK FB_SolSpringPiston_2Pos
(* Single-solenoid, spring-return 2-position actuator.
   Coil energised  -> drives to EXTENDED.
   Coil de-energised -> mechanical spring returns to RETRACTED.

   The coil is a continuous force against the spring, so Section 2 uses a
   LATCH-and-RETAIN pattern: the coil is set TRUE on Extend command and
   FALSE on Retract command, and RETAINS its state (via VAR_OUTPUT retain)
   any cycle no explicit command is active. Without the latch the coil
   would drop the moment the extended sensor fires and the spring would
   immediately pull the piston back.

   Fail-safe by construction: broken wire, dead coil, PLC power loss
   or e-stop all leave bOutSolenoid FALSE and the spring retracts.

   Interface is kept symmetric with FB_SolSolPiston_2Pos so a sequencer FB
   (e.g. FB_PistonAutoCycle) can drive either actuator type without a
   custom variant. Reuses ST_HmiPiston unchanged; the retract-coil mirror
   field (stHmi.bOutSolenoidRetract) is always FALSE because no retract
   coil exists on this actuator. *)
VAR_INPUT
    (* Automatic Commands from PLC sequence logic. Wired to FALSE in MAIN until FB_Auto exists. *)
    bAutoCmdExtend    : BOOL;
    bAutoCmdRetract   : BOOL;

    (* External jog request (e.g. panel push-button). OR-merged with the
       HMI's stHmi.bManJogExtend inside so a physical PB and the HMI
       button can drive the same jog without stepping on each other.
       Only takes effect while eMode = Manual (same gate as the HMI jog).

       MOMENTARY, unlike the HMI jog: holding energises the coil, RELEASING
       de-energises it and the spring returns the piston. The panel has no
       jog-retract button, so a latching PB would strand the piston extended
       until someone walked to the HMI. The HMI jog keeps its latching
       behaviour because bManJogRetract sits right next to it. *)
    bJogExtend        : BOOL;


    (* Physical Feedback (Proximity Switches) *)
    bSwitchExtended   : BOOL;
    bSwitchRetracted  : BOOL;
END_VAR

VAR_IN_OUT
    (* HMI contract — mode, manual + simulate inputs, latched + sensor status *)
    stHmi             : ST_HmiPiston;
END_VAR

VAR_OUTPUT
    (* Physical Output to Solenoid — SINGLE coil.
       TRUE  = coil energised, actuator drives EXTENDED.
       FALSE = coil de-energised, spring returns actuator to RETRACTED. *)
    bOutSolenoid      : BOOL;
END_VAR

VAR
    (* Internal Target States *)
    bTargetExtend     : BOOL;
    bTargetRetract    : BOOL;

    (* HMI Manual-Button Edge Detection *)
    fbTrigManExtend   : R_TRIG;
    fbTrigManRetract  : R_TRIG;

    (* Falling edge of bJogExtend = the panel push-button was released.
       Needed because Section 2 retains the coil when no branch matches, so
       without an explicit release edge a momentary PB would latch the
       piston extended with no panel-side way to bring it back. *)
    fbTrigJogRelease  : F_TRIG;

    (* Effective sensor states = real OR HMI simulate. Recomputed every cycle in Section 0a. *)
    bSwitchExtended_eff  : BOOL;
    bSwitchRetracted_eff : BOOL;

    (* Previous-cycle snapshots for the mode-field bridge in Section 0b.
       Classic PLC HMI writes stHmi.bMode (Rotary Switch is boolean-only);
       web HMI writes stHmi.eMode (enum via ToggleSwitch). This FB is the
       authoritative reader of eMode, so we sync in whichever direction
       changed since last cycle. *)
    bPrevMode : BOOL;
    ePrevMode : E_ControlMode;
END_VAR

(* ==========================================
   0b. MODE-FIELD BRIDGE — sync bMode <-> eMode
   The classic PLC HMI (VISUs) writes stHmi.bMode because its Rotary Switch
   element is boolean-only. FlowerPyHmi writes stHmi.eMode over ADS.
   (The retired Flower_HMI web project did the same via a ToggleSwitch.) Rest of this FB reads eMode as the authoritative field,
   so we mirror bMode into eMode when the classic HMI toggled the switch,
   and mirror eMode back into bMode when the web HMI (or anyone else) wrote
   eMode. Edge-triggered — whichever side changed since last cycle wins.
   Runs BEFORE Section 0 so downstream logic sees a coherent eMode.
   ========================================== *)
IF stHmi.bMode <> bPrevMode THEN
    // Classic VISU changed bMode → propagate to eMode
    IF stHmi.bMode THEN
        stHmi.eMode := E_ControlMode.Automatic;
    ELSE
        stHmi.eMode := E_ControlMode.Manual;
    END_IF;
ELSIF stHmi.eMode <> ePrevMode THEN
    // Web HMI (or any other writer) changed eMode → propagate to bMode
    stHmi.bMode := (stHmi.eMode = E_ControlMode.Automatic);
END_IF;

bPrevMode := stHmi.bMode;
ePrevMode := stHmi.eMode;

(* ==========================================
   0a. EFFECTIVE SENSOR INPUTS (real OR HMI simulate)
   ========================================== *)
bSwitchExtended_eff  := bSwitchExtended  OR stHmi.bSimulateExtended;
bSwitchRetracted_eff := bSwitchRetracted OR stHmi.bSimulateRetracted;

(* ==========================================
   0. HMI MANUAL BUTTON LATCHING (Radio-Button Behavior)
   ========================================== *)
fbTrigManExtend(CLK := stHmi.bManCmdExtend);
fbTrigManRetract(CLK := stHmi.bManCmdRetract);

// Independent IFs (not ELSIF): if multiple edges fire in the same cycle, the last one wins (Retract > Extend).
IF fbTrigManExtend.Q  THEN stHmi.bSelectedExtend := TRUE;  stHmi.bSelectedRetract := FALSE; END_IF;
IF fbTrigManRetract.Q THEN stHmi.bSelectedExtend := FALSE; stHmi.bSelectedRetract := TRUE;  END_IF;

IF stHmi.eMode = E_ControlMode.Automatic THEN
    stHmi.bSelectedExtend := FALSE; stHmi.bSelectedRetract := FALSE;
END_IF;

(* ==========================================
   1. MODE SELECTION & COMMAND MAPPING
   Spring-return semantics: both bAutoCmd* inputs are accepted for interface
   parity with FB_SolSolPiston_2Pos, but physically only Extend commands the
   coil. If both auto bits are TRUE we treat it as a conflict and de-energise
   (safe default — spring retracts).
   ========================================== *)
IF stHmi.eMode = E_ControlMode.Automatic THEN
    bTargetExtend  := bAutoCmdExtend  AND NOT bAutoCmdRetract;
    bTargetRetract := bAutoCmdRetract AND NOT bAutoCmdExtend;

ELSIF stHmi.eMode = E_ControlMode.Manual THEN
    bTargetExtend  := stHmi.bSelectedExtend;
    bTargetRetract := stHmi.bSelectedRetract;

ELSE
    // Safe default: undefined mode → no targets
    bTargetExtend  := FALSE;
    bTargetRetract := FALSE;
END_IF;

(* ==========================================
   1a. JOG OVERRIDE — clear latched selection while either jog is held
   ========================================== *)
// Section 1 above already copied stHmi.bSelected* into bTarget*. The stale
// bTarget* is harmless because Section 2's jog branches sit ahead of the
// bTarget* branches in the IF/ELSIF ladder and preempt them.
IF stHmi.bManJogExtend OR stHmi.bManJogRetract OR bJogExtend THEN
    stHmi.bSelectedExtend := FALSE; stHmi.bSelectedRetract := FALSE;
END_IF;

(* ==========================================
   1b. TARGET-REACHED RESET — clear bSelected* once the piston arrives
   ========================================== *)
IF stHmi.bSelectedExtend  AND bSwitchExtended_eff  THEN stHmi.bSelectedExtend  := FALSE; END_IF;
IF stHmi.bSelectedRetract AND bSwitchRetracted_eff THEN stHmi.bSelectedRetract := FALSE; END_IF;

(* ==========================================
   1c. PANEL JOG RELEASE EDGE
   Called unconditionally so the edge is never missed. MAIN gates bJogExtend
   with bManualMode, so this also pulses on a Manual -> Auto switch; Section 2
   gates the release branch on Manual, and MAIN forces eMode to Automatic
   BEFORE calling this FB, so that pulse is correctly ignored and the master
   cycle's retract states take the piston home instead.
   ========================================== *)
fbTrigJogRelease(CLK := bJogExtend);

(* ==========================================
   2. SOLENOID CONTROL — single coil, LATCH-and-RETAIN
   The coil is a continuous force against the spring. If it drops, the spring
   wins and the actuator retracts. So the coil must be LATCHED TRUE from the
   moment Extend is commanded until Retract is commanded — not pulsed until
   the sensor fires (which is the double-solenoid pattern).
   Structure:
     - Jog branches first, gated by Manual mode.
     - Then the panel-jog RELEASE edge, which is the one exception to the
       retain rule: the PB is momentary, so letting go must drive the coil
       FALSE instead of letting it latch. The HMI jog is NOT momentary --
       it latches, because bManJogRetract exists to undo it.
     - Explicit Extend / Retract command branches drive the coil to a
       definite state.
     - The IF ladder has NO ELSE. When no branch matches, VAR_OUTPUT retain
       semantics carry the coil forward:
         * At the Extended sensor after a successful extend (Section 1b just
           cleared bTargetExtend) → coil retains TRUE → piston HOLDS.
         * At the Retracted sensor after a successful retract → coil retains
           FALSE → piston HOLDS retracted (spring already there).
         * Sequencer DWELL_EXT (both auto bits FALSE) → coil retains TRUE
           for the full dwell instead of releasing the piston.
     - No sensor guards on the drive branches: holding the coil TRUE while
       at the Extended sensor is normal operation, not a wasted drive.
   Fail-safe still holds: cold boot, PLC reset, or e-stop leave bOutSolenoid
   at its default FALSE and the spring retracts.
   ========================================== *)
// JOG EXTEND: while held in Manual, energise coil. HMI-owned bManJogExtend
// OR external bJogExtend (panel push-button) -- both share the Manual gate.
IF (stHmi.bManJogExtend OR bJogExtend) AND stHmi.eMode = E_ControlMode.Manual THEN
    bOutSolenoid := TRUE;

// JOG RETRACT: while held in Manual, de-energise coil (spring retracts)
ELSIF stHmi.bManJogRetract AND stHmi.eMode = E_ControlMode.Manual THEN
    bOutSolenoid := FALSE;

// PANEL JOG RELEASE: the PB is momentary, so letting go must send the piston
// home rather than leaving the coil latched by the retain rule below.
// Position in the ladder is deliberate:
//   - AFTER both jog branches, so if the HMI jog-extend is still held the
//     coil stays TRUE and this one-scan pulse is simply ignored;
//   - BEFORE the bTarget branches, so a latched HMI Extend selection cannot
//     re-energise the coil the instant the operator lets go. Section 1a
//     already cleared bSelected* while the jog was held, so this only
//     reinforces the same intent.
ELSIF fbTrigJogRelease.Q AND stHmi.eMode = E_ControlMode.Manual THEN
    bOutSolenoid := FALSE;

// EXTEND commanded — energise coil (latched via retain when bTargetExtend clears)
ELSIF bTargetExtend THEN
    bOutSolenoid := TRUE;

// RETRACT commanded — de-energise coil, spring retracts
ELSIF bTargetRetract THEN
    bOutSolenoid := FALSE;

// No branch → bOutSolenoid RETAINS its previous value (see block header).
END_IF;

(* ==========================================
   3. HMI STATUS FEEDBACK
   bIsMoving is derived from sensor state alone: with Section 2's latch
   semantics, bOutSolenoid stays TRUE at the extended limit — so ORing
   it in would report "moving" while the piston is actually parked.
   "Between the two limits" is accurate for both strokes: coil-driven
   extend and spring-driven retract both traverse that gap.

   bOutSolenoidRetract is written FALSE unconditionally — no retract coil
   exists on a spring-return actuator, so the mirror stays cleared.
   ========================================== *)
stHmi.bIsExtended         := bSwitchExtended_eff;
stHmi.bIsRetracted        := bSwitchRetracted_eff;
stHmi.bIsMoving           := NOT bSwitchExtended_eff AND NOT bSwitchRetracted_eff;
stHmi.bOutSolenoidExtend  := bOutSolenoid;
stHmi.bOutSolenoidRetract := FALSE;

END_FUNCTION_BLOCK

// ---- POUs/FB_MasterAutoCycle.TcPOU
FUNCTION_BLOCK FB_MasterAutoCycle
(* Full-machine coordinated auto sequence spanning the robot and the 3
   pairs of SepSol / PushSol pistons (pair count fixed at 3 for this
   machine).

   Robot interface (TCP-only, 2026-07-26). The former discrete-I/O handshake
   is retired. All robot-side signals travel over FB_RobotTcpClient's
   STATE:n / CMD:n protocol:

     Robot -> PLC   nRobotCmd in {1,2}  (1=start, 2=reset error)
                    MAIN R_TRIGs on the edges; start pulse arrives here as
                    the VAR_INPUT bExtStartPulse.
     PLC -> Robot   nStateOut = TO_INT(eStep) or MANUAL(30)
                    Written by MAIN each scan, pushed by FB_RobotTcpClient
                    on change and as keep-alive.

   TWO KINDS OF START, WITH DIFFERENT OWNERS (2026-07-29):

     Operator START  = "home the pistons and arm the machine".
                       stHmi.bStart, from the HMI button or the green PB3 in
                       Automatic. Runs the INIT retract chain and stops in IDLE.
                       It does NOT run a bulb cycle.
     Robot CMD:1     = "run one bulb cycle". Arrives as bExtStartPulse. Valid
                       only from IDLE, i.e. only once a human has armed the
                       machine. bSimStartAssembly is its bench stand-in.

   So the machine cannot move after a power cycle, after Manual, or after a
   STOP until an operator presses START; and once armed, only the robot decides
   when a bulb runs. bContinuous is gone entirely (2026-08-06) -- it was written
   force-clears it every scan) -- it was the last path that could start motion
   with nothing external gating it.

   BENCH-BUILD EXCEPTION (2026-08-13, gated 2026-08-17): bTempTestContinuesAutoRun
   deliberately re-opens exactly that path, for log-file soak testing. It is kept
   for reuse on the next project rather than deleted, and it is therefore gated
   behind the VAR CONSTANT bBenchBuild, which is FALSE in any build that goes on
   a machine. Read bBenchBuild's comment before changing either.

   Sequence (all 3 Sep/Push pairs move in parallel; both grips move together):

     NOT_HOMED               In Automatic, NOT armed. Entered on power-up (the
                             declared default of stHmi.eStep), on any time in
                             Manual, and on operator STOP. Reports STATE:40,
                             which the robot reads as "wait". Exits only on
                             operator START -> INIT chain, bHomeThenIdle TRUE.
     IDLE                    Armed. Any of bExtStartPulse (robot CMD:1, and also
                             how the PB2+PB3 operator hold arrives), bStartCycle
                             (operator "run one bulb" from an HMI), bSimStartAssembly
                             (bench stand-in for the robot) or SimIdle -> INIT chain
                             with bHomeThenIdle FALSE (a bulb cycle). Four ways in,
                             logged distinctly so the ring says which.
                             Operator START here is IGNORED (2026-08-05).
                             It used to re-home and come back, which was a no-op
                             in outcome and let a green-before-orange press of
                             the PB2+PB3 combo lose its bulb request: the combo's
                             one-scan pulse landed mid INIT_* chain, where
                             nothing consumes it. Section 0b logs the refusal.
     INIT_PUSH_RETRACTING    drive PushCmdRetract[1..3]; wait AND of all
                             PushIsRetracted. Guarantees pistons are home before
                             a cycle starts, even if a prior manual move left
                             them extended.
     INIT_SEP_RETRACTING     drive SepCmdRetract[1..3]; wait AND of all
                             SepIsRetracted. Push must retract first (see INIT
                             above) because sep retract with push extended is
                             the same collision case avoided end-of-cycle.
     INIT_GRIP_RETRACTING    drive GripCmdRetract[1..2]; wait bGripIsRetracted[1]
                             OR [2] -- the same OR deviation as the two GRIP
                             states below, so error 8 shares their blind spot:
                             it fires only if BOTH grippers fail to come home.
                             Defensive symmetry with the INIT
                             Sep/Push states, so a manual jog left extended
                             does not collide with the arriving plate.
                             THE ONE PLACE THE TWO CALLERS DIVERGE: exits to
                             IDLE when bHomeThenIdle, else to CHECK_PLATE.
     CHECK_PLATE              wait bPlateOk = bPlateSenL OR bPlateSenR (robot
                             has placed the plate on the fixture). OR, not AND:
                             only one plate sensor is confirmed wired, so an AND
                             would fault every cycle. Deliberate field deviation
                             -- see the plate/grip note in CLAUDE.md before
                             "fixing" it. Latched at start only;
                             sensors are not monitored past this step.
                             stCfg.bBypassPlateSensors removes the timeout
                             ERROR only -- the sensor fast-path still applies,
                             and on expiry the cycle continues instead of
                             raising error 9. bNoSensors does NOT cover this
                             state.
     GRIP_EXTENDING          drive GripCmdExtend[1..2]; wait bGripIsExtended[1]
                             OR [2] -- again OR, not AND, because GripSolR has
                             no air on the machine. COST: with either sensor
                             satisfying it, a genuine single-gripper failure is
                             invisible and the cycle can run on a plate clamped
                             from one side; error 10 fires only if BOTH fail.
     SEP_EXTENDING           drive SepCmdExtend[1..3]; wait AND of all SepIsExtended.
                             Grip stays extended for every state below.
     PUSH_EXTENDING          drive PushCmdExtend[1..3]; wait AND of all PushIsExtended
     DWELL_PUSH              hold both extended; wait tDwellPushMs
     PUSH_RETRACTING         drive PushCmdRetract[1..3]; wait AND of all PushIsRetracted
     PUSH_RETRACTED_DWELL    wait tPushRetractedDwellMs
     SEP_RETRACTING          drive SepCmdRetract[1..3]; wait AND of all SepIsRetracted
     SEP_RETRACTED_DWELL     wait tSepRetractedDwellMs
     GRIP_RETRACTING         drive GripCmdRetract[1..2]; wait bGripIsRetracted[1]
                             OR [2] (same OR deviation as GRIP_EXTENDING, and
                             error 11 has the same blind spot). Releases the
                             plate; increment nCyclesCompleted; back to IDLE --
                             still armed, so the robot's next CMD:1 runs another.
     ERR                     latched; iErrorCode set to step code. Reports
                             STATE:99, on which the robot answers CMD:2. RESET
                             (that CMD:2, the HMI button, or the orange PB2)
                             clears the error and enters the RECOVER_* chain
                             below -- NOT the INIT chain, and NOT straight to
                             IDLE. A fault leaves the pistons anywhere, so
                             advertising IDLE(0) would claim ready while it is
                             not, and RESET landing in IDLE with the robot still
                             asking made RESET itself a start button.
     RECOVER_PUSH_RETR       Fault-recovery retract chain (50/51/52), added
     RECOVER_SEP_RETR        2026-08-05. Same motion and the same collision
     RECOVER_GRIP_RETR       ordering as the INIT chain, but its own identity so
                             a failed RECOVERY is distinguishable from a failed
                             ARMING: error codes 12/13/14 instead of 6/7/8, and
                             its own sStepText. Entered ONLY from ERR on RESET.
                             RECOVER_GRIP_RETR always exits to IDLE -- by then
                             the machine really is homed, so reporting STATE:0 is
                             honest. The robot needed no new branch: it acts on 0
                             and 99 and treats everything else as "wait".

   Error codes:
     0  = OK
     1  = SEP_EXTENDING timed out
     3  = PUSH_EXTENDING timed out
     4  = PUSH_RETRACTING timed out
     5  = SEP_RETRACTING timed out
     6  = INIT_PUSH_RETRACTING timed out
     7  = INIT_SEP_RETRACTING timed out
     8  = INIT_GRIP_RETRACTING timed out
     9  = CHECK_PLATE timed out (plate never arrived / one sensor never TRUE)
          -- suppressed while stCfg.bBypassPlateSensors is set
    10  = GRIP_EXTENDING timed out
    11  = GRIP_RETRACTING timed out
    12  = RECOVER_PUSH_RETR timed out  -- recovery, deliberately distinct from 6
    13  = RECOVER_SEP_RETR timed out   -- distinct from 7
    14  = RECOVER_GRIP_RETR timed out  -- distinct from 8
    99  = RETIRED (was 'Operator STOP while running'). STOP now disarms to
          NOT_HOMED instead of faulting -- see Section 2. Do not reuse the
          number: old log entries and CSV exports still carry it.

   The former WAIT_POS2 state (error code 2) is retired: the robot code
   (src0.lua PerformStandSequence) already moves the arm clear of the
   stand BEFORE raising STAND_SEQ_DO, so the PLC does not need a separate
   "robot moved away" wait between SEP_EXTENDING and PUSH_EXTENDING. The
   E_MasterAutoStep.WAIT_POS2 enum value and stHmi.bSimStep_WaitPos2 flag
   remain declared but are unused; safe to remove once the HMI is cleaned.

   Per-step Sim flags on stHmi (bSimStep_Idle, bSimStep_SepExt, and so on)
   let a bench operator advance any waiting step without physical sensors.
   Rising-edge triggered; the FB auto-clears the flag after consumption.

